KUKA KRL program: MyProgram_119().src

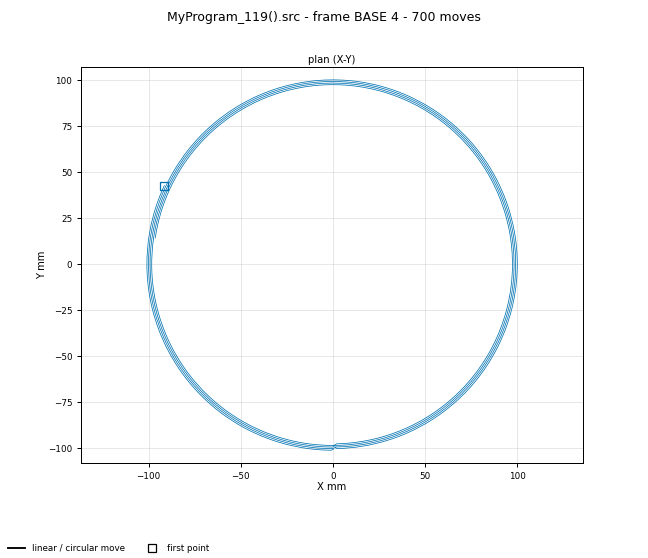
[picture p0: tool path of MyProgram_119().src in frame BASE 4, 700 of 700 moves have a stored position in this frame; points joined in program order, loops and branches not executed]
&ACCESS RVP
&REL 1
&PARAM TEMPLATE = C:\KRC\Roboter\Template\vorgabe
&PARAM EDITMASK = *
DEF MyProgram_119()
; ---- Setting reference (Base) ----
$BASE = BASE_DATA[4]

; --------------------------
; ---- Setting tool (TCP) ----
$TOOL = TOOL_DATA[3]
; --------------------------

$VEL.CP = VEL_APROX_PRINT
Startdeposition()
$VEL.CP = VEL_PRINT
LIN {X -91.493,Y 42.7067,Z 101,A 150.6977,B 24.9258,C -1.9891,E1 24.8544,E2 294.7155} C_DIS
LIN {X -92.8066,Y 39.7749,Z 101,A 152.6178,B 24.926,C -1.9868,E1 24.8522,E2 292.79} C_DIS
LIN {X -93.9596,Y 36.9649,Z 101,A 154.2845,B 24.9265,C -1.9796,E1 24.8505,E2 291.1312} C_DIS
LIN {X -95.1822,Y 33.6934,Z 101,A 156.3544,B 24.9268,C -1.9765,E1 24.8485,E2 289.0571} C_DIS
LIN {X -96.2277,Y 30.5829,Z 101,A 158.5957,B 24.9262,C -1.9837,E1 24.8466,E2 286.7858} C_DIS
LIN {X -97.2713,Y 27.0799,Z 101,A 160.5089,B 24.9271,C -1.9716,E1 24.8451,E2 284.8903} C_DIS
LIN {X -98.522,Y 22.1039,Z 101,A 163.2579,B 24.9282,C -1.9568,E1 24.8434,E2 282.1606} C_DIS
LIN {X -99.102,Y 19.3303,Z 101,A 165.2055,B 24.9277,C -1.9633,E1 24.8423,E2 280.1859} C_DIS
LIN {X -99.9373,Y 14.4011,Z 101,A 167.61,B 24.9295,C -1.9393,E1 24.8413,E2 277.8242} C_DIS
LIN {X -100.2963,Y 11.6391,Z 101,A 169.6473,B 24.9287,C -1.9499,E1 24.8406,E2 275.7496} C_DIS
LIN {X -100.8986,Y 3.8154,Z 101,A 173.661,B 24.9309,C -1.9204,E1 24.8399,E2 271.782} C_DIS
LIN {X -100.9502,Y -1.9696,Z 101,A 177.1716,B 24.9311,C -1.9176,E1 24.8399,E2 268.257} C_DIS
LIN {X -100.7114,Y -7.2249,Z 101,A 179.6583,B 24.933,C -1.891,E1 24.8402,E2 265.8188} C_DIS
LIN {X -100.1169,Y -13.0935,Z 101,A -176.3946,B 24.9323,C -1.9008,E1 24.8414,E2 261.8247} C_DIS
LIN {X -99.4794,Y -17.292,Z 101,A -174.1202,B 24.9331,C -1.8886,E1 24.8424,E2 259.566} C_DIS
LIN {X -98.8843,Y -20.4137,Z 101,A -172.2959,B 24.9335,C -1.8837,E1 24.8434,E2 257.7426} C_DIS
LIN {X -98.0917,Y -23.9337,Z 101,A -170.2804,B 24.934,C -1.8763,E1 24.8447,E2 255.733} C_DIS
LIN {X -97.2543,Y -27.1399,Z 101,A -168.3863,B 24.9344,C -1.871,E1 24.8461,E2 253.8404} C_DIS
LIN {X -95.3072,Y -33.3371,Z 101,A -164.6672,B 24.9351,C -1.8611,E1 24.8493,E2 250.1237} C_DIS
LIN {X -93.8132,Y -37.3364,Z 101,A -162.0084,B 24.935,C -1.8621,E1 24.852,E2 247.4474} C_DIS
LIN {X -91.5082,Y -42.6739,Z 101,A -158.9614,B 24.9363,C -1.844,E1 24.8554,E2 244.427} C_DIS
LIN {X -89.9932,Y -45.7829,Z 101,A -156.9304,B 24.9365,C -1.8409,E1 24.8579,E2 242.3925} C_DIS
LIN {X -88.288,Y -48.9909,Z 101,A -154.8266,B 24.9368,C -1.8367,E1 24.8607,E2 240.2874} C_DIS
LIN {X -85.444,Y -53.7984,Z 101,A -151.8215,B 24.9377,C -1.8226,E1 24.865,E2 237.3006} C_DIS
LIN {X -83.1904,Y -57.2225,Z 101,A -149.2876,B 24.9377,C -1.8239,E1 24.869,E2 234.751} C_DIS
LIN {X -81.3627,Y -59.7909,Z 101,A -147.5016,B 24.938,C -1.8194,E1 24.8719,E2 232.967} C_DIS
LIN {X -79.3097,Y -62.4885,Z 101,A -145.5763,B 24.9383,C -1.8148,E1 24.8752,E2 231.0434} C_DIS
LIN {X -77.0494,Y -65.2555,Z 101,A -143.6749,B 24.9389,C -1.8056,E1 24.8785,E2 229.1552} C_DIS
LIN {X -73.7308,Y -68.983,Z 101,A -140.7273,B 24.939,C -1.8033,E1 24.8841,E2 226.1999} C_DIS
LIN {X -71.3796,Y -71.4151,Z 101,A -138.9011,B 24.9396,C -1.7959,E1 24.8876,E2 224.3837} C_DIS
LIN {X -69.3421,Y -73.393,Z 101,A -137.1004,B 24.9393,C -1.7993,E1 24.8913,E2 222.5673} C_DIS
LIN {X -66.913,Y -75.6161,Z 101,A -134.6373,B 24.9381,C -1.817,E1 24.8966,E2 220.0524} C_DIS
LIN {X -63.8127,Y -78.2486,Z 101,A -132.5208,B 24.9389,C -1.8058,E1 24.9011,E2 217.9546} C_DIS
LIN {X -61.117,Y -80.3733,Z 101,A -131.0124,B 24.9402,C -1.7864,E1 24.9043,E2 216.4868} C_DIS
LIN {X -58.1677,Y -82.5329,Z 101,A -128.8413,B 24.9402,C -1.7864,E1 24.9093,E2 214.3081} C_DIS
LIN {X -54.8555,Y -84.7693,Z 101,A -126.6695,B 24.9407,C -1.7793,E1 24.9143,E2 212.146} C_DIS
LIN {X -50.7449,Y -87.292,Z 101,A -123.4729,B 24.9398,C -1.7921,E1 24.9221,E2 208.9093} C_DIS
LIN {X -47.8522,Y -88.9106,Z 101,A -121.9794,B 24.9409,C -1.7754,E1 24.9257,E2 207.4513} C_DIS
LIN {X -45.4378,Y -90.1696,Z 101,A -120.33,B 24.9409,C -1.7772,E1 24.9298,E2 205.7931} C_DIS
LIN {X -41.9811,Y -91.8297,Z 101,A -118.2406,B 24.9412,C -1.7715,E1 24.935,E2 203.712} C_DIS
LIN {X -38.9897,Y -93.1379,Z 101,A -116.4085,B 24.9414,C -1.7688,E1 24.9397,E2 201.882} C_DIS
LIN {X -34.2328,Y -94.9895,Z 101,A -113.3032,B 24.941,C -1.7739,E1 24.9479,E2 198.7582} C_DIS
LIN {X -30.1552,Y -96.3615,Z 101,A -111.3711,B 24.9424,C -1.7531,E1 24.9529,E2 196.872} C_DIS
LIN {X -26.5243,Y -97.4234,Z 101,A -108.3775,B 24.9404,C -1.7833,E1 24.9612,E2 193.8019} C_DIS
LIN {X -22.855,Y -98.3488,Z 101,A -106.897,B 24.9421,C -1.7571,E1 24.965,E2 192.3815} C_DIS
LIN {X -16.9752,Y -99.5327,Z 101,A -103.5642,B 24.9424,C -1.7531,E1 24.9742,E2 189.0547} C_DIS
LIN {X -13.0619,Y -100.121,Z 101,A -101.1076,B 24.9419,C -1.7605,E1 24.981,E2 186.5785} C_DIS
LIN {X -9.5303,Y -100.5189,Z 101,A -99.1069,B 24.9419,C -1.7597,E1 24.9865,E2 184.5785} C_DIS
LIN {X -5.5002,Y -100.8195,Z 101,A -96.5488,B 24.9413,C -1.7698,E1 24.9937,E2 181.9954} C_DIS
LIN {X -0.9129,Y -100.9657,Z 101,A -94.2262,B 24.942,C -1.7595,E1 25.0002,E2 179.6972} C_DIS
LIN {X -0.9129,Y -100.9657,Z 101,A -94.2262,B 24.942,C -1.7595,E1 25.0002,E2 179.6972} C_DIS
Enddeposition()
LIN {X 0.7006,Y -100.097,Z 101,A -94.1894,B 24.9431,C -1.7417,E1 25.0002,E2 179.7026} C_DIS
Startdeposition()
$VEL.CP = VEL_PRINT
LIN {X -2.9837,Y -100.0551,Z 101,A -96.3968,B 24.9434,C -1.7377,E1 24.9939,E2 181.9196} C_DIS
LIN {X -8.2546,Y -99.759,Z 101,A -99.1397,B 24.9427,C -1.748,E1 24.9864,E2 184.6391} C_DIS
LIN {X -10.6456,Y -99.5321,Z 101,A -100.6356,B 24.943,C -1.7436,E1 24.9822,E2 186.1463} C_DIS
LIN {X -16.0258,Y -98.8096,Z 101,A -104.2786,B 24.9443,C -1.7247,E1 24.972,E2 189.8371} C_DIS
LIN {X -19.3833,Y -98.2058,Z 101,A -105.6359,B 24.9428,C -1.7472,E1 24.9684,E2 191.1426} C_DIS
LIN {X -21.9592,Y -97.663,Z 101,A -107.9018,B 24.9445,C -1.7203,E1 24.9621,E2 193.4751} C_DIS
LIN {X -25.8197,Y -96.7127,Z 101,A -109.6986,B 24.9433,C -1.739,E1 24.9573,E2 195.2303} C_DIS
LIN {X -30.2063,Y -95.435,Z 101,A -112.2271,B 24.943,C -1.7439,E1 24.9506,E2 197.7513} C_DIS
LIN {X -35.0024,Y -93.7802,Z 101,A -115.2233,B 24.943,C -1.7432,E1 24.9427,E2 200.7553} C_DIS
LIN {X -39.1334,Y -92.1335,Z 101,A -117.5532,B 24.9424,C -1.7534,E1 24.9367,E2 203.066} C_DIS
LIN {X -42.6063,Y -90.5803,Z 101,A -119.8193,B 24.9424,C -1.7527,E1 24.9309,E2 205.3393} C_DIS
LIN {X -45.6761,Y -89.0709,Z 101,A -121.6953,B 24.9421,C -1.7581,E1 24.9263,E2 207.2076} C_DIS
LIN {X -48.5502,Y -87.5379,Z 101,A -124.3798,B 24.9438,C -1.7317,E1 24.9195,E2 209.9625} C_DIS
LIN {X -52.3977,Y -85.2915,Z 101,A -126.098,B 24.9416,C -1.7646,E1 24.9156,E2 211.6076} C_DIS
LIN {X -55.2394,Y -83.4779,Z 101,A -128.0767,B 24.9416,C -1.7659,E1 24.9109,E2 213.5897} C_DIS
LIN {X -57.5637,Y -81.8939,Z 101,A -129.9662,B 24.942,C -1.7588,E1 24.9066,E2 215.5026} C_DIS
LIN {X -60.5866,Y -79.6839,Z 101,A -132.7293,B 24.9432,C -1.741,E1 24.9003,E2 218.3179} C_DIS
LIN {X -64.2306,Y -76.7742,Z 101,A -134.8539,B 24.9416,C -1.7649,E1 24.8958,E2 220.3938} C_DIS
LIN {X -67.9037,Y -73.5466,Z 101,A -137.4269,B 24.9407,C -1.7782,E1 24.8905,E2 222.9453} C_DIS
LIN {X -70.1968,Y -71.3609,Z 101,A -139.231,B 24.9405,C -1.7823,E1 24.8869,E2 224.7471} C_DIS
LIN {X -72.61,Y -68.9051,Z 101,A -141.3632,B 24.9405,C -1.781,E1 24.8828,E2 226.8917} C_DIS
LIN {X -76.3774,Y -64.703,Z 101,A -144.5016,B 24.9398,C -1.7915,E1 24.877,E2 230.0192} C_DIS
LIN {X -78.6568,Y -61.9118,Z 101,A -146.6049,B 24.9396,C -1.795,E1 24.8733,E2 232.124} C_DIS
LIN {X -80.6494,Y -59.2928,Z 101,A -148.3867,B 24.9391,C -1.8031,E1 24.8703,E2 233.8951} C_DIS
LIN {X -82.5834,Y -56.5702,Z 101,A -150.8268,B 24.9399,C -1.79,E1 24.8664,E2 236.3785} C_DIS
LIN {X -84.496,Y -53.671,Z 101,A -152.1216,B 24.938,C -1.8186,E1 24.8645,E2 237.6116} C_DIS
LIN {X -86.627,Y -50.1577,Z 101,A -154.4412,B 24.9375,C -1.826,E1 24.8612,E2 239.9256} C_DIS
LIN {X -88.6618,Y -46.4655,Z 101,A -157.1228,B 24.9377,C -1.8234,E1 24.8576,E2 242.6275} C_DIS
LIN {X -90.0555,Y -43.7045,Z 101,A -159.0063,B 24.9377,C -1.8245,E1 24.8553,E2 244.5186} C_DIS
LIN {X -91.9197,Y -39.634,Z 101,A -162.5269,B 24.9393,C -1.7999,E1 24.8513,E2 248.1171} C_DIS
LIN {X -93.9682,Y -34.4956,Z 101,A -165.82,B 24.9389,C -1.8051,E1 24.8481,E2 251.4166} C_DIS
LIN {X -95.8576,Y -28.8337,Z 101,A -167.8821,B 24.9351,C -1.8603,E1 24.8465,E2 253.3587} C_DIS
LIN {X -96.5103,Y -26.569,Z 101,A -169.4978,B 24.9355,C -1.8555,E1 24.8452,E2 254.9954} C_DIS
LIN {X -97.3864,Y -23.155,Z 101,A -171.6399,B 24.9353,C -1.8575,E1 24.8438,E2 257.1453} C_DIS
LIN {X -98.2035,Y -19.3963,Z 101,A -173.8412,B 24.9348,C -1.8644,E1 24.8425,E2 259.3431} C_DIS
LIN {X -98.8363,Y -15.862,Z 101,A -176.063,B 24.9348,C -1.8653,E1 24.8415,E2 261.576} C_DIS
LIN {X -99.2655,Y -12.8949,Z 101,A -178.3144,B 24.9356,C -1.8531,E1 24.8407,E2 263.87} C_DIS
LIN {X -99.7582,Y -8.2647,Z 101,A -179.9211,B 24.9326,C -1.8966,E1 24.8403,E2 265.3825} C_DIS
LIN {X -100.0729,Y -2.3714,Z 101,A 175.9269,B 24.9336,C -1.8817,E1 24.8398,E2 269.595} C_DIS
LIN {X -100.0954,Y 0.9959,Z 101,A 174.3514,B 24.9324,C -1.8995,E1 24.8398,E2 271.1374} C_DIS
LIN {X -99.9873,Y 4.7622,Z 101,A 171.7367,B 24.9329,C -1.8914,E1 24.8401,E2 273.7873} C_DIS
LIN {X -99.7433,Y 8.4515,Z 101,A 169.9451,B 24.9317,C -1.9089,E1 24.8405,E2 275.548} C_DIS
LIN {X -99.2648,Y 12.9005,Z 101,A 167.5862,B 24.9306,C -1.9238,E1 24.8413,E2 277.8853} C_DIS
LIN {X -98.8225,Y 15.9485,Z 101,A 165.8016,B 24.9303,C -1.9287,E1 24.842,E2 279.6688} C_DIS
LIN {X -97.8958,Y 20.8933,Z 101,A 162.6806,B 24.9302,C -1.93,E1 24.8437,E2 282.8052} C_DIS
LIN {X -96.9348,Y 24.9712,Z 101,A 160.2729,B 24.9296,C -1.9373,E1 24.8454,E2 285.2096} C_DIS
LIN {X -95.5364,Y 29.8792,Z 101,A 157.2634,B 24.9292,C -1.9435,E1 24.8478,E2 288.2216} C_DIS
LIN {X -93.8825,Y 34.7305,Z 101,A 154.4878,B 24.9281,C -1.9579,E1 24.8503,E2 290.9787} C_DIS
LIN {X -92.1093,Y 39.1904,Z 101,A 151.9333,B 24.927,C -1.9727,E1 24.853,E2 293.5121} C_DIS
LIN {X -91.0749,Y 41.539,Z 101,A 150.4396,B 24.9268,C -1.9763,E1 24.8547,E2 295.0054} C_DIS
LIN {X -89.832,Y 44.1616,Z 101,A 148.0741,B 24.9281,C -1.9579,E1 24.8577,E2 297.4276} C_DIS
LIN {X -88.0636,Y 47.5894,Z 101,A 145.8824,B 24.9276,C -1.9649,E1 24.8606,E2 299.6142} C_DIS
LIN {X -86.2144,Y 50.8626,Z 101,A 144.331,B 24.9257,C -1.991,E1 24.8627,E2 301.1113} C_DIS
LIN {X -84.1782,Y 54.1661,Z 101,A 141.6968,B 24.9262,C -1.9835,E1 24.8666,E2 303.7768} C_DIS
LIN {X -80.2524,Y 59.8291,Z 101,A 137.9554,B 24.9249,C -2.0011,E1 24.8727,E2 307.4945} C_DIS
LIN {X -77.5079,Y 63.3449,Z 101,A 135.1326,B 24.9251,C -1.9988,E1 24.8776,E2 310.3361} C_DIS
LIN {X -73.9412,Y 67.4737,Z 101,A 132.0295,B 24.9244,C -2.0074,E1 24.8834,E2 313.4326} C_DIS
LIN {X -71.0995,Y 70.4614,Z 101,A 129.7788,B 24.9237,C -2.0168,E1 24.8877,E2 315.6704} C_DIS
LIN {X -67.7192,Y 73.7159,Z 101,A 127.0704,B 24.9233,C -2.0224,E1 24.8932,E2 318.3767} C_DIS
LIN {X -63.4929,Y 77.3882,Z 101,A 124.1903,B 24.9219,C -2.0406,E1 24.8993,E2 321.2246} C_DIS
LIN {X -61.4928,Y 78.9855,Z 101,A 122.181,B 24.9231,C -2.0252,E1 24.9038,E2 323.278} C_DIS
LIN {X -57.0068,Y 82.281,Z 101,A 119.1357,B 24.9222,C -2.0365,E1 24.9107,E2 326.307} C_DIS
LIN {X -53.02,Y 84.9047,Z 101,A 116.1874,B 24.9224,C -2.0342,E1 24.9177,E2 329.2701} C_DIS
LIN {X -50.0776,Y 86.673,Z 101,A 114.506,B 24.9214,C -2.0475,E1 24.9217,E2 330.925} C_DIS
LIN {X -46.541,Y 88.622,Z 101,A 112.3664,B 24.9206,C -2.0573,E1 24.9269,E2 333.0472} C_DIS
LIN {X -43.3756,Y 90.2135,Z 101,A 110.3409,B 24.9204,C -2.0607,E1 24.9319,E2 335.0701} C_DIS
LIN {X -39.8894,Y 91.8083,Z 101,A 107.6228,B 24.9215,C -2.0457,E1 24.939,E2 337.8301} C_DIS
LIN {X -36.6127,Y 93.1635,Z 101,A 106.2301,B 24.9196,C -2.0707,E1 24.9425,E2 339.1665} C_DIS
LIN {X -34.1586,Y 94.0911,Z 101,A 104.5603,B 24.9199,C -2.0668,E1 24.9469,E2 340.8491} C_DIS
LIN {X -31.2828,Y 95.0871,Z 101,A 103.0132,B 24.9192,C -2.0757,E1 24.9509,E2 342.3778} C_DIS
LIN {X -29.0314,Y 95.799,Z 101,A 101.4147,B 24.9198,C -2.0685,E1 24.9552,E2 343.9962} C_DIS
LIN {X -25.7437,Y 96.7332,Z 101,A 98.9755,B 24.9209,C -2.0536,E1 24.9619,E2 346.4746} C_DIS
LIN {X -22.1291,Y 97.6237,Z 101,A 97.5469,B 24.9188,C -2.0803,E1 24.9656,E2 347.8415} C_DIS
LIN {X -16.5738,Y 98.7179,Z 101,A 94.1038,B 24.9192,C -2.0757,E1 24.9751,E2 351.2994} C_DIS
LIN {X -10.1902,Y 99.5798,Z 101,A 90.7337,B 24.9181,C -2.0893,E1 24.9844,E2 354.6397} C_DIS
LIN {X -4.7667,Y 99.9871,Z 101,A 87.5182,B 24.9183,C -2.0868,E1 24.9934,E2 357.8622} C_DIS
LIN {X 0.5268,Y 100.0982,Z 101,A 84.3427,B 24.9187,C -2.0823,E1 25.0022,E2 361.0486} C_DIS
LIN {X 5.7674,Y 99.9336,Z 101,A 81.4712,B 24.9183,C -2.0873,E1 25.0102,E2 363.9076} C_DIS
LIN {X 8.3217,Y 99.7536,Z 101,A 79.1426,B 24.9207,C -2.0558,E1 25.0169,E2 366.3096} C_DIS
LIN {X 12.5536,Y 99.3097,Z 101,A 77.3041,B 24.9191,C -2.077,E1 25.0219,E2 368.0964} C_DIS
LIN {X 17.1869,Y 98.6145,Z 101,A 74.8657,B 24.9185,C -2.0851,E1 25.0285,E2 370.5131} C_DIS
LIN {X 22.4978,Y 97.5386,Z 101,A 71.4561,B 24.9195,C -2.0723,E1 25.0379,E2 373.9488} C_DIS
LIN {X 25.2776,Y 96.8561,Z 101,A 69.9253,B 24.9192,C -2.0753,E1 25.042,E2 375.4703} C_DIS
LIN {X 28.795,Y 95.8691,Z 101,A 67.4467,B 24.9205,C -2.0594,E1 25.0487,E2 377.9821} C_DIS
LIN {X 31.9491,Y 94.864,Z 101,A 65.7801,B 24.9199,C -2.0663,E1 25.0531,E2 379.6292} C_DIS
LIN {X 35.3881,Y 93.6355,Z 101,A 63.9232,B 24.9194,C -2.0731,E1 25.0579,E2 381.4662} C_DIS
LIN {X 38.949,Y 92.2112,Z 101,A 61.8875,B 24.9191,C -2.0768,E1 25.0632,E2 383.4884} C_DIS
LIN {X 41.1192,Y 91.2641,Z 101,A 60.5769,B 24.9191,C -2.077,E1 25.0665,E2 384.7954} C_DIS
LIN {X 43.6247,Y 90.0938,Z 101,A 58.7276,B 24.92,C -2.065,E1 25.0712,E2 386.6683} C_DIS
LIN {X 49.68,Y 86.9015,Z 101,A 54.9069,B 24.9202,C -2.0634,E1 25.0806,E2 390.4819} C_DIS
LIN {X 52.4585,Y 85.2543,Z 101,A 53.0967,B 24.9202,C -2.0621,E1 25.0849,E2 392.2895} C_DIS
LIN {X 54.5736,Y 83.9166,Z 101,A 51.4144,B 24.9212,C -2.0503,E1 25.0889,E2 393.9942} C_DIS
LIN {X 57.9099,Y 81.6483,Z 101,A 49.2842,B 24.9209,C -2.0533,E1 25.0938,E2 396.11} C_DIS
LIN {X 60.6655,Y 79.6236,Z 101,A 46.6029,B 24.9233,C -2.0222,E1 25.0999,E2 398.8552} C_DIS
LIN {X 64.1859,Y 76.8125,Z 101,A 44.8781,B 24.9212,C -2.05,E1 25.1034,E2 400.5077} C_DIS
LIN {X 66.6943,Y 74.6445,Z 101,A 42.9433,B 24.9216,C -2.0448,E1 25.1075,E2 402.4471} C_DIS
LIN {X 69.2792,Y 72.2522,Z 101,A 40.8642,B 24.9221,C -2.0382,E1 25.1118,E2 404.5332} C_DIS
LIN {X 71.9424,Y 69.6006,Z 101,A 38.7499,B 24.9223,C -2.035,E1 25.1159,E2 406.646} C_DIS
LIN {X 74.5803,Y 66.766,Z 101,A 36.5814,B 24.9226,C -2.0319,E1 25.12,E2 408.8123} C_DIS
LIN {X 76.207,Y 64.9031,Z 101,A 35.1815,B 24.9228,C -2.0293,E1 25.1225,E2 410.2122} C_DIS
LIN {X 78.6359,Y 61.9382,Z 101,A 33.0135,B 24.9231,C -2.0251,E1 25.1263,E2 412.38} C_DIS
LIN {X 80.7719,Y 59.1254,Z 101,A 30.763,B 24.9242,C -2.0111,E1 25.1301,E2 414.6527} C_DIS
LIN {X 83.494,Y 55.2149,Z 101,A 28.2001,B 24.9242,C -2.0106,E1 25.1341,E2 417.2041} C_DIS
LIN {X 85.5275,Y 52.0093,Z 101,A 26.0772,B 24.9245,C -2.0069,E1 25.1373,E2 419.3251} C_DIS
LIN {X 88.4343,Y 46.8975,Z 101,A 23.0136,B 24.9243,C -2.0097,E1 25.1414,E2 422.3661} C_DIS
LIN {X 90.4834,Y 42.8137,Z 101,A 19.9323,B 24.9262,C -1.9839,E1 25.1453,E2 425.4917} C_DIS
LIN {X 92.813,Y 37.4932,Z 101,A 17.0107,B 24.9257,C -1.9903,E1 25.1485,E2 428.3822} C_DIS
LIN {X 93.702,Y 35.2126,Z 101,A 15.3498,B 24.9268,C -1.9759,E1 25.1501,E2 430.068} C_DIS
LIN {X 94.8531,Y 31.9815,Z 101,A 13.5164,B 24.9268,C -1.9752,E1 25.1518,E2 431.8926} C_DIS
LIN {X 95.8353,Y 28.909,Z 101,A 11.2507,B 24.9285,C -1.9529,E1 25.1537,E2 434.198} C_DIS
LIN {X 97.7108,Y 21.7417,Z 101,A 7.6499,B 24.9276,C -1.9654,E1 25.1561,E2 437.7486} C_DIS
LIN {X 98.5163,Y 17.7329,Z 101,A 4.7673,B 24.9297,C -1.9364,E1 25.1577,E2 440.6826} C_DIS
LIN {X 99.0662,Y 14.3483,Z 101,A 2.5039,B 24.931,C -1.9183,E1 25.1586,E2 442.9755} C_DIS
LIN {X 99.5773,Y 10.2143,Z 101,A 1.336,B 24.928,C -1.9594,E1 25.1589,E2 444.0395} C_DIS
LIN {X 99.9111,Y 6.1631,Z 101,A -1.9506,B 24.9314,C -1.9133,E1 25.1596,E2 447.4153} C_DIS
LIN {X 100.0566,Y 2.9338,Z 101,A -3.848,B 24.9319,C -1.9055,E1 25.1598,E2 449.3198} C_DIS
LIN {X 100.0978,Y -0.6116,Z 101,A -5.3962,B 24.931,C -1.9182,E1 25.1598,E2 450.8289} C_DIS
LIN {X 100.0063,Y -4.3206,Z 101,A -7.9573,B 24.9328,C -1.8939,E1 25.1595,E2 453.4321} C_DIS
LIN {X 99.7945,Y -7.8104,Z 101,A -10.2974,B 24.9342,C -1.8739,E1 25.159,E2 455.8054} C_DIS
LIN {X 99.3001,Y -12.6283,Z 101,A -13.3909,B 24.9357,C -1.8523,E1 25.1578,E2 458.9317} C_DIS
LIN {X 98.3394,Y -18.6906,Z 101,A -15.4002,B 24.9323,C -1.901,E1 25.1569,E2 460.8144} C_DIS
LIN {X 97.2465,Y -23.7283,Z 101,A -18.6275,B 24.9337,C -1.8804,E1 25.155,E2 464.0716} C_DIS
LIN {X 96.3574,Y -27.1146,Z 101,A -21.8325,B 24.9375,C -1.8262,E1 25.1525,E2 467.3858} C_DIS
LIN {X 94.4759,Y -33.0791,Z 101,A -24.151,B 24.9348,C -1.8652,E1 25.1505,E2 469.5995} C_DIS
LIN {X 93.3391,Y -36.1656,Z 101,A -27.1789,B 24.9383,C -1.8138,E1 25.1473,E2 472.7318} C_DIS
LIN {X 91.0143,Y -41.6735,Z 101,A -29.3314,B 24.9356,C -1.8538,E1 25.145,E2 474.7781} C_DIS
LIN {X 89.3765,Y -45.0782,Z 101,A -32.0583,B 24.9376,C -1.8248,E1 25.1415,E2 477.5589} C_DIS
LIN {X 87.8167,Y -48.0446,Z 101,A -33.8804,B 24.9377,C -1.823,E1 25.1391,E2 479.3757} C_DIS
LIN {X 85.0848,Y -52.7316,Z 101,A -36.3481,B 24.9366,C -1.8395,E1 25.1357,E2 481.7918} C_DIS
LIN {X 82.1303,Y -57.2236,Z 101,A -39.399,B 24.9371,C -1.8319,E1 25.131,E2 484.8456} C_DIS
LIN {X 79.0604,Y -61.3964,Z 101,A -42.4573,B 24.9379,C -1.82,E1 25.1259,E2 487.9171} C_DIS
LIN {X 77.261,Y -63.6452,Z 101,A -44.5001,B 24.9393,C -1.8,E1 25.1222,E2 489.9977} C_DIS
LIN {X 74.6432,Y -66.6958,Z 101,A -46.5022,B 24.9389,C -1.8059,E1 25.1185,E2 491.9769} C_DIS
LIN {X 71.8665,Y -69.6793,Z 101,A -48.7723,B 24.9391,C -1.8026,E1 25.1142,E2 494.245} C_DIS
LIN {X 67.9034,Y -73.5469,Z 101,A -52.0245,B 24.9398,C -1.7917,E1 25.1076,E2 497.5094} C_DIS
LIN {X 65.5412,Y -75.6596,Z 101,A -54.039,B 24.9406,C -1.7796,E1 25.1033,E2 499.5444} C_DIS
LIN {X 61.9682,Y -78.6122,Z 101,A -57.3523,B 24.9427,C -1.7481,E1 25.096,E2 502.9197} C_DIS
LIN {X 57.8656,Y -81.6799,Z 101,A -58.7583,B 24.9392,C -1.8016,E1 25.0931,E2 504.1944} C_DIS
LIN {X 53.1117,Y -84.8474,Z 101,A -62.5262,B 24.9409,C -1.7755,E1 25.0842,E2 508.0115} C_DIS
LIN {X 50.3503,Y -86.5163,Z 101,A -64.7948,B 24.9422,C -1.7557,E1 25.0787,E2 510.3199} C_DIS
LIN {X 43.8916,Y -89.9656,Z 101,A -68.6624,B 24.9419,C -1.7611,E1 25.0691,E2 514.1639} C_DIS
LIN {X 38.9198,Y -92.2235,Z 101,A -72.2976,B 24.9435,C -1.7369,E1 25.0597,E2 517.8477} C_DIS
LIN {X 35.4642,Y -93.6067,Z 101,A -73.8684,B 24.9423,C -1.7553,E1 25.0557,E2 519.3713} C_DIS
LIN {X 32.0718,Y -94.8226,Z 101,A -77.1878,B 24.9455,C -1.7051,E1 25.0467,E2 522.803} C_DIS
LIN {X 25.9246,Y -96.6844,Z 101,A -79.6063,B 24.9427,C -1.7485,E1 25.0405,E2 525.1149} C_DIS
LIN {X 19.2144,Y -98.2386,Z 101,A -83.3099,B 24.9423,C -1.7539,E1 25.0304,E2 528.8007} C_DIS
LIN {X 12.1755,Y -99.3578,Z 101,A -87.46,B 24.9427,C -1.7482,E1 25.0189,E2 532.9603} C_DIS
LIN {X 5.8421,Y -99.9294,Z 101,A -91.7549,B 24.9444,C -1.722,E1 25.0068,E2 537.3153} C_DIS
LIN {X 2.2509,Y -100.0751,Z 101,A -93.3016,B 24.9432,C -1.7403,E1 25.0026,E2 538.8183} C_DIS
LIN {X 2.2509,Y -100.0751,Z 101,A -93.3016,B 24.9432,C -1.7403,E1 25.0026,E2 538.8183} C_DIS
Enddeposition()
LIN {X 0.6916,Y -99.2244,Z 101,A -93.6165,B 24.9408,C -1.7769,E1 25.002,E2 539.0464} C_DIS
Startdeposition()
$VEL.CP = VEL_PRINT
LIN {X 6.3538,Y -99.0267,Z 101,A -89.6742,B 24.9391,C -1.8033,E1 25.0131,E2 535.0428} C_DIS
LIN {X 12.1636,Y -98.4832,Z 101,A -86.8433,B 24.9403,C -1.7847,E1 25.0209,E2 532.2576} C_DIS
LIN {X 18.1451,Y -97.5584,Z 101,A -83.2608,B 24.9399,C -1.7906,E1 25.0308,E2 528.6648} C_DIS
LIN {X 23.6602,Y -96.3678,Z 101,A -80.0271,B 24.9398,C -1.7927,E1 25.0396,E2 525.4304} C_DIS
LIN {X 26.8003,Y -95.5424,Z 101,A -78.3328,B 24.9401,C -1.7878,E1 25.0441,E2 523.7505} C_DIS
LIN {X 31.9669,Y -93.9401,Z 101,A -74.9259,B 24.9391,C -1.8024,E1 25.0533,E2 520.3154} C_DIS
LIN {X 35.8208,Y -92.54,Z 101,A -71.783,B 24.9368,C -1.8358,E1 25.0617,E2 517.1001} C_DIS
LIN {X 40.3117,Y -90.6739,Z 101,A -69.7341,B 24.9386,C -1.8103,E1 25.0667,E2 515.1166} C_DIS
LIN {X 43.8065,Y -89.0372,Z 101,A -67.6711,B 24.9388,C -1.8074,E1 25.0719,E2 513.0657} C_DIS
LIN {X 45.9989,Y -87.9245,Z 101,A -66.2309,B 24.9385,C -1.8106,E1 25.0755,E2 511.6219} C_DIS
LIN {X 50.5879,Y -85.3664,Z 101,A -63.1025,B 24.9379,C -1.8198,E1 25.0831,E2 508.4812} C_DIS
LIN {X 55.554,Y -82.221,Z 101,A -59.8303,B 24.9379,C -1.8216,E1 25.0908,E2 505.2155} C_DIS
LIN {X 58.3914,Y -80.2313,Z 101,A -57.2713,B 24.936,C -1.8478,E1 25.0967,E2 502.6036} C_DIS
LIN {X 61.312,Y -78.0221,Z 101,A -55.6812,B 24.9371,C -1.8315,E1 25.1001,E2 501.0577} C_DIS
LIN {X 63.2853,Y -76.43,Z 101,A -53.8126,B 24.9358,C -1.8509,E1 25.1042,E2 499.1506} C_DIS
LIN {X 65.8199,Y -74.2598,Z 101,A -52.4995,B 24.9372,C -1.8309,E1 25.1068,E2 497.8899} C_DIS
LIN {X 69.8907,Y -70.4406,Z 101,A -49.0231,B 24.9359,C -1.8486,E1 25.1139,E2 494.3859} C_DIS
LIN {X 74.0098,Y -66.0992,Z 101,A -46.0025,B 24.9365,C -1.84,E1 25.1196,E2 491.399} C_DIS
LIN {X 77.5141,Y -61.9549,Z 101,A -42.4986,B 24.9349,C -1.8629,E1 25.1259,E2 487.8571} C_DIS
LIN {X 80.3128,Y -58.2802,Z 101,A -39.8563,B 24.9345,C -1.8691,E1 25.1303,E2 485.2127} C_DIS
LIN {X 82.4339,Y -55.2397,Z 101,A -37.3834,B 24.9331,C -1.8885,E1 25.1343,E2 482.7063} C_DIS
LIN {X 85.1675,Y -50.9244,Z 101,A -34.228,B 24.9319,C -1.9053,E1 25.1389,E2 479.5273} C_DIS
LIN {X 87.1332,Y -47.4804,Z 101,A -32.9116,B 24.9343,C -1.8727,E1 25.1406,E2 478.2946} C_DIS
LIN {X 88.6335,Y -44.6207,Z 101,A -30.6535,B 24.9328,C -1.894,E1 25.1435,E2 475.9982} C_DIS
LIN {X 90.1198,Y -41.5343,Z 101,A -28.7669,B 24.9326,C -1.8963,E1 25.1457,E2 474.1164} C_DIS
LIN {X 90.9993,Y -39.5686,Z 101,A -26.9002,B 24.9305,C -1.9254,E1 25.1479,E2 472.1913} C_DIS
LIN {X 92.5514,Y -35.7918,Z 101,A -25.096,B 24.9316,C -1.9101,E1 25.1497,E2 470.4331} C_DIS
LIN {X 93.7134,Y -32.6251,Z 101,A -22.5669,B 24.9294,C -1.9399,E1 25.152,E2 467.848} C_DIS
LIN {X 95.0254,Y -28.5807,Z 101,A -20.7534,B 24.9308,C -1.9215,E1 25.1535,E2 466.0883} C_DIS
LIN {X 96.026,Y -25.0129,Z 101,A -18.7831,B 24.9308,C -1.9215,E1 25.1549,E2 464.1295} C_DIS
LIN {X 96.6333,Y -22.5519,Z 101,A -16.8022,B 24.9289,C -1.9471,E1 25.1562,E2 462.0995} C_DIS
LIN {X 97.3395,Y -19.2831,Z 101,A -15.3945,B 24.93,C -1.932,E1 25.157,E2 460.7356} C_DIS
LIN {X 98.2316,Y -14.0393,Z 101,A -12.2896,B 24.9292,C -1.9432,E1 25.1584,E2 457.6224} C_DIS
LIN {X 98.6678,Y -10.5476,Z 101,A -10.5648,B 24.9296,C -1.9374,E1 25.1589,E2 455.9216} C_DIS
LIN {X 98.9435,Y -7.5412,Z 101,A -7.7728,B 24.9261,C -1.9856,E1 25.1596,E2 453.0325} C_DIS
LIN {X 99.1809,Y -3.1146,Z 101,A -6.001,B 24.9278,C -1.9618,E1 25.1598,E2 451.3274} C_DIS
LIN {X 99.1866,Y 2.929,Z 101,A -1.8322,B 24.925,C -2.0006,E1 25.1596,E2 447.0918} C_DIS
LIN {X 98.9706,Y 7.1841,Z 101,A 0.0102,B 24.9262,C -1.9834,E1 25.1592,E2 445.301} C_DIS
LIN {X 98.1834,Y 14.3784,Z 101,A 4.8169,B 24.9233,C -2.0221,E1 25.1575,E2 440.4314} C_DIS
LIN {X 97.4534,Y 18.6917,Z 101,A 6.5866,B 24.925,C -1.9993,E1 25.1567,E2 438.7256} C_DIS
LIN {X 96.75,Y 22.0468,Z 101,A 8.4021,B 24.925,C -1.9989,E1 25.1556,E2 436.9218} C_DIS
LIN {X 95.7769,Y 25.9485,Z 101,A 10.8729,B 24.9241,C -2.012,E1 25.1539,E2 434.4343} C_DIS
LIN {X 94.8252,Y 29.2361,Z 101,A 12.8188,B 24.9237,C -2.0168,E1 25.1523,E2 432.4882} C_DIS
LIN {X 93.8389,Y 32.2656,Z 101,A 14.7723,B 24.923,C -2.0268,E1 25.1506,E2 430.5221} C_DIS
LIN {X 92.5015,Y 35.9189,Z 101,A 16.6628,B 24.9236,C -2.0192,E1 25.1488,E2 428.6601} C_DIS
LIN {X 90.6665,Y 40.3278,Z 101,A 20.0236,B 24.9211,C -2.0512,E1 25.145,E2 425.242} C_DIS
LIN {X 88.5403,Y 44.8031,Z 101,A 22.5888,B 24.9214,C -2.0474,E1 25.1419,E2 422.6995} C_DIS
LIN {X 87.0559,Y 47.6229,Z 101,A 24.6266,B 24.9204,C -2.0603,E1 25.1391,E2 420.642} C_DIS
LIN {X 84.739,Y 51.632,Z 101,A 26.9269,B 24.921,C -2.0526,E1 25.1359,E2 418.3717} C_DIS
LIN {X 82.719,Y 54.8101,Z 101,A 29.0185,B 24.9208,C -2.055,E1 25.1327,E2 416.285} C_DIS
LIN {X 80.146,Y 58.5079,Z 101,A 31.7329,B 24.92,C -2.066,E1 25.1283,E2 413.5579} C_DIS
LIN {X 77.8797,Y 61.4922,Z 101,A 33.7179,B 24.92,C -2.0642,E1 25.125,E2 411.5865} C_DIS
LIN {X 75.911,Y 63.9093,Z 101,A 35.5946,B 24.9195,C -2.0714,E1 25.1216,E2 409.7013} C_DIS
LIN {X 74.3224,Y 65.75,Z 101,A 37.1035,B 24.919,C -2.0787,E1 25.1188,E2 408.182} C_DIS
LIN {X 72.0836,Y 68.1952,Z 101,A 39.0416,B 24.9186,C -2.0839,E1 25.1151,E2 406.24} C_DIS
LIN {X 69.5519,Y 70.7753,Z 101,A 41.1003,B 24.9183,C -2.0873,E1 25.111,E2 404.1822} C_DIS
LIN {X 66.9465,Y 73.2444,Z 101,A 43.1126,B 24.9181,C -2.0892,E1 25.1069,E2 402.1736} C_DIS
LIN {X 64.2983,Y 75.5796,Z 101,A 44.9423,B 24.9185,C -2.0851,E1 25.1031,E2 400.3607} C_DIS
LIN {X 61.0442,Y 78.2337,Z 101,A 47.66,B 24.9172,C -2.1009,E1 25.0971,E2 397.6159} C_DIS
LIN {X 57.9902,Y 80.5225,Z 101,A 49.7483,B 24.9172,C -2.1003,E1 25.0925,E2 395.5365} C_DIS
LIN {X 55.4221,Y 82.3104,Z 101,A 51.6178,B 24.9168,C -2.1057,E1 25.0881,E2 393.6605} C_DIS
LIN {X 52.9337,Y 83.933,Z 101,A 53.3745,B 24.9165,C -2.1099,E1 25.084,E2 391.8994} C_DIS
LIN {X 49.5448,Y 85.976,Z 101,A 55.2659,B 24.9174,C -2.0983,E1 25.0795,E2 390.0414} C_DIS
LIN {X 45.8575,Y 87.9989,Z 101,A 58.0416,B 24.9161,C -2.1148,E1 25.0726,E2 387.2347} C_DIS
LIN {X 42.9669,Y 89.4449,Z 101,A 59.7167,B 24.9165,C -2.1098,E1 25.0685,E2 385.5757} C_DIS
LIN {X 40.1177,Y 90.76,Z 101,A 61.6838,B 24.9159,C -2.1177,E1 25.0634,E2 383.5948} C_DIS
LIN {X 35.9128,Y 92.5039,Z 101,A 64.3228,B 24.9156,C -2.1208,E1 25.0566,E2 380.9544} C_DIS
LIN {X 32.6977,Y 93.688,Z 101,A 66.9189,B 24.9136,C -2.146,E1 25.0496,E2 378.304} C_DIS
LIN {X 28.5833,Y 95.0246,Z 101,A 68.7127,B 24.9156,C -2.1213,E1 25.045,E2 376.5719} C_DIS
LIN {X 25.5467,Y 95.8855,Z 101,A 70.5042,B 24.9156,C -2.1213,E1 25.0402,E2 374.7831} C_DIS
LIN {X 23.2273,Y 96.4734,Z 101,A 71.8399,B 24.9156,C -2.1204,E1 25.0365,E2 373.4516} C_DIS
LIN {X 19.4176,Y 97.3129,Z 101,A 74.2357,B 24.9152,C -2.1268,E1 25.03,E2 371.0438} C_DIS
LIN {X 15.8591,Y 97.9556,Z 101,A 76.7431,B 24.9139,C -2.1431,E1 25.023,E2 368.5002} C_DIS
LIN {X 12.4184,Y 98.4502,Z 101,A 78.364,B 24.915,C -2.1292,E1 25.0186,E2 366.9135} C_DIS
LIN {X 7.0075,Y 98.9825,Z 101,A 81.1509,B 24.916,C -2.1166,E1 25.0109,E2 364.1583} C_DIS
LIN {X 1.3541,Y 99.2216,Z 101,A 84.4602,B 24.9159,C -2.1178,E1 25.0017,E2 360.847} C_DIS
LIN {X -4.3687,Y 99.1336,Z 101,A 87.472,B 24.9168,C -2.1063,E1 24.9934,E2 357.8622} C_DIS
LIN {X -9.2517,Y 98.7976,Z 101,A 90.7224,B 24.9157,C -2.1203,E1 24.9842,E2 354.5773} C_DIS
LIN {X -14.0161,Y 98.2349,Z 101,A 93.5781,B 24.9156,C -2.1217,E1 24.9763,E2 351.7162} C_DIS
LIN {X -18.1165,Y 97.5636,Z 101,A 96.4336,B 24.9144,C -2.1363,E1 24.9683,E2 348.8232} C_DIS
LIN {X -21.3424,Y 96.9076,Z 101,A 97.7828,B 24.9161,C -2.1149,E1 24.9648,E2 347.5232} C_DIS
LIN {X -25.0619,Y 96.0134,Z 101,A 100.0596,B 24.9161,C -2.1152,E1 24.9586,E2 345.2425} C_DIS
LIN {X -28.7965,Y 94.9614,Z 101,A 102.5226,B 24.9157,C -2.1206,E1 24.9519,E2 342.7625} C_DIS
LIN {X -32.7072,Y 93.6846,Z 101,A 104.8611,B 24.916,C -2.1164,E1 24.9458,E2 340.4296} C_DIS
LIN {X -36.3507,Y 92.3319,Z 101,A 107.4865,B 24.9152,C -2.1269,E1 24.9389,E2 337.7736} C_DIS
LIN {X -39.6612,Y 90.9589,Z 101,A 108.9927,B 24.917,C -2.1041,E1 24.9351,E2 336.3183} C_DIS
LIN {X -42.4708,Y 89.6833,Z 101,A 111.0187,B 24.9165,C -2.1099,E1 24.9299,E2 334.2734} C_DIS
LIN {X -45.9858,Y 87.9314,Z 101,A 113.1082,B 24.9173,C -2.0999,E1 24.9248,E2 332.2019} C_DIS
LIN {X -48.7251,Y 86.444,Z 101,A 114.8934,B 24.9176,C -2.0963,E1 24.9204,E2 330.4202} C_DIS
LIN {X -53.1742,Y 83.7813,Z 101,A 117.9615,B 24.9178,C -2.0933,E1 24.9131,E2 327.3496} C_DIS
LIN {X -56.1482,Y 81.8185,Z 101,A 120.2897,B 24.9174,C -2.0987,E1 24.9077,E2 325.0009} C_DIS
LIN {X -61.7314,Y 77.6907,Z 101,A 123.9325,B 24.9191,C -2.0776,E1 24.8997,E2 321.3952} C_DIS
LIN {X -64.2208,Y 75.6457,Z 101,A 126.0114,B 24.9188,C -2.081,E1 24.8952,E2 319.3003} C_DIS
LIN {X -67.0993,Y 73.1042,Z 101,A 128.0301,B 24.9197,C -2.0691,E1 24.891,E2 317.3018} C_DIS
LIN {X -69.5965,Y 70.7312,Z 101,A 130.2343,B 24.9195,C -2.0717,E1 24.8866,E2 315.0822} C_DIS
LIN {X -72.5465,Y 67.703,Z 101,A 133.0859,B 24.9189,C -2.0797,E1 24.881,E2 312.1992} C_DIS
LIN {X -74.931,Y 65.0536,Z 101,A 135.4065,B 24.9186,C -2.0835,E1 24.8768,E2 309.8591} C_DIS
LIN {X -77.8049,Y 61.5869,Z 101,A 137.1334,B 24.9214,C -2.0468,E1 24.8739,E2 308.2114} C_DIS
LIN {X -81.0438,Y 57.2582,Z 101,A 140.4455,B 24.9216,C -2.0448,E1 24.8684,E2 304.8883} C_DIS
LIN {X -84.4996,Y 52.0259,Z 101,A 144.1518,B 24.9222,C -2.0374,E1 24.8628,E2 301.1807} C_DIS
LIN {X -86.4907,Y 48.6414,Z 101,A 147.2761,B 24.9204,C -2.06,E1 24.8584,E2 297.9862} C_DIS
LIN {X -88.9227,Y 44.0374,Z 101,A 149.3298,B 24.9236,C -2.0188,E1 24.8559,E2 296.0199} C_DIS
LIN {X -90.4317,Y 40.8491,Z 101,A 151.3862,B 24.924,C -2.0133,E1 24.8535,E2 293.9653} C_DIS
LIN {X -92.7186,Y 35.3533,Z 101,A 154.8262,B 24.9248,C -2.0029,E1 24.8499,E2 290.531} C_DIS
LIN {X -94.8443,Y 29.1746,Z 101,A 158.642,B 24.9256,C -1.9925,E1 24.8465,E2 286.7182} C_DIS
LIN {X -95.7548,Y 26.0305,Z 101,A 160.8806,B 24.9251,C -1.9982,E1 24.8448,E2 284.4529} C_DIS
LIN {X -96.9395,Y 21.196,Z 101,A 163.7449,B 24.9258,C -1.9887,E1 24.843,E2 281.5944} C_DIS
LIN {X -97.836,Y 16.5744,Z 101,A 166.1852,B 24.9272,C -1.9707,E1 24.8418,E2 279.1827} C_DIS
LIN {X -98.3354,Y 13.3046,Z 101,A 168.1772,B 24.9274,C -1.9673,E1 24.841,E2 277.187} C_DIS
LIN {X -98.7235,Y 10.0156,Z 101,A 170.0014,B 24.9281,C -1.9582,E1 24.8405,E2 275.3735} C_DIS
LIN {X -99.042,Y 6.1268,Z 101,A 172.2309,B 24.9287,C -1.9501,E1 24.84,E2 273.1499} C_DIS
LIN {X -99.1915,Y 2.768,Z 101,A 174.358,B 24.9287,C -1.9501,E1 24.8398,E2 271.01} C_DIS
LIN {X -99.2287,Y -0.4872,Z 101,A 176.3263,B 24.9289,C -1.947,E1 24.8398,E2 269.0372} C_DIS
LIN {X -99.0715,Y -5.6035,Z 101,A 179.0811,B 24.9301,C -1.9308,E1 24.8401,E2 266.3045} C_DIS
LIN {X -98.7771,Y -9.4735,Z 101,A -178.1706,B 24.9294,C -1.9407,E1 24.8408,E2 263.516} C_DIS
LIN {X -98.4142,Y -12.6963,Z 101,A -177.1328,B 24.9318,C -1.9068,E1 24.8411,E2 262.5531} C_DIS
LIN {X -98.0471,Y -15.2749,Z 101,A -175.2845,B 24.9314,C -1.9135,E1 24.8419,E2 260.6776} C_DIS
LIN {X -97.5178,Y -18.357,Z 101,A -173.3544,B 24.9314,C -1.9121,E1 24.8428,E2 258.7396} C_DIS
LIN {X -96.7804,Y -21.9152,Z 101,A -171.2355,B 24.9319,C -1.9063,E1 24.8441,E2 256.6221} C_DIS
LIN {X -95.9715,Y -25.2251,Z 101,A -169.2467,B 24.9323,C -1.9009,E1 24.8455,E2 254.6344} C_DIS
LIN {X -95.0127,Y -28.6236,Z 101,A -166.6437,B 24.9313,C -1.9139,E1 24.8476,E2 251.9853} C_DIS
LIN {X -93.8293,Y -32.2898,Z 101,A -164.9883,B 24.9332,C -1.888,E1 24.849,E2 250.3825} C_DIS
LIN {X -92.6985,Y -35.4063,Z 101,A -163.3101,B 24.9341,C -1.8743,E1 24.8506,E2 248.7273} C_DIS
LIN {X -90.9835,Y -39.6049,Z 101,A -160.4627,B 24.9341,C -1.8745,E1 24.8537,E2 245.8637} C_DIS
LIN {X -89.5953,Y -42.6539,Z 101,A -158.4712,B 24.9344,C -1.871,E1 24.856,E2 243.8698} C_DIS
LIN {X -88.1041,Y -45.6565,Z 101,A -156.4916,B 24.9347,C -1.8671,E1 24.8586,E2 241.8888} C_DIS
LIN {X -86.5603,Y -48.5169,Z 101,A -154.801,B 24.9355,C -1.8557,E1 24.8608,E2 240.2166} C_DIS
LIN {X -84.6236,Y -51.8218,Z 101,A -152.3532,B 24.9353,C -1.8579,E1 24.8643,E2 237.7508} C_DIS
LIN {X -81.9341,Y -55.9778,Z 101,A -149.5094,B 24.9358,C -1.85,E1 24.8687,E2 234.9115} C_DIS
LIN {X -80.1354,Y -58.5225,Z 101,A -147.7543,B 24.9363,C -1.844,E1 24.8716,E2 233.1621} C_DIS
LIN {X -77.4904,Y -61.9848,Z 101,A -145.1959,B 24.9366,C -1.8394,E1 24.876,E2 230.6025} C_DIS
LIN {X -75.579,Y -64.299,Z 101,A -142.6043,B 24.9348,C -1.8654,E1 24.8808,E2 227.9372} C_DIS
LIN {X -72.2921,Y -67.9735,Z 101,A -140.6224,B 24.9373,C -1.8288,E1 24.8844,E2 226.0338} C_DIS
LIN {X -69.7037,Y -70.6253,Z 101,A -138.4997,B 24.9377,C -1.8237,E1 24.8886,E2 223.9143} C_DIS
LIN {X -66.8615,Y -73.3224,Z 101,A -136.285,B 24.9381,C -1.8174,E1 24.8931,E2 221.7055} C_DIS
LIN {X -64.6554,Y -75.2749,Z 101,A -134.1342,B 24.9372,C -1.8299,E1 24.8977,E2 219.5165} C_DIS
LIN {X -60.0562,Y -78.9944,Z 101,A -131.0058,B 24.9384,C -1.8135,E1 24.9045,E2 216.4156} C_DIS
LIN {X -58.0196,Y -80.5015,Z 101,A -129.4374,B 24.9383,C -1.8148,E1 24.9081,E2 214.8387} C_DIS
LIN {X -53.2839,Y -83.7109,Z 101,A -126.1864,B 24.9388,C -1.8077,E1 24.9156,E2 211.594} C_DIS
LIN {X -49.0631,Y -86.2527,Z 101,A -123.527,B 24.9395,C -1.7969,E1 24.922,E2 208.952} C_DIS
LIN {X -46.5781,Y -87.6194,Z 101,A -121.8164,B 24.9395,C -1.7974,E1 24.9262,E2 207.2355} C_DIS
LIN {X -44.0863,Y -88.8985,Z 101,A -120.2311,B 24.9397,C -1.7942,E1 24.9301,E2 205.6535} C_DIS
LIN {X -41.0855,Y -90.3252,Z 101,A -118.0237,B 24.9391,C -1.8024,E1 24.9358,E2 203.4211} C_DIS
LIN {X -37.4294,Y -91.8998,Z 101,A -115.8956,B 24.9397,C -1.7939,E1 24.9412,E2 201.3084} C_DIS
LIN {X -31.965,Y -93.9407,Z 101,A -112.5499,B 24.9399,C -1.7901,E1 24.95,E2 197.9651} C_DIS
LIN {X -28.8738,Y -94.9375,Z 101,A -110.6482,B 24.9399,C -1.7896,E1 24.9551,E2 196.0612} C_DIS
LIN {X -26.599,Y -95.599,Z 101,A -109.342,B 24.9402,C -1.7865,E1 24.9586,E2 194.7602} C_DIS
LIN {X -22.6931,Y -96.6007,Z 101,A -106.9386,B 24.9401,C -1.7879,E1 24.9651,E2 192.35} C_DIS
LIN {X -19.4121,Y -97.314,Z 101,A -105.1829,B 24.9406,C -1.7804,E1 24.9699,E2 190.6102} C_DIS
LIN {X -16.0922,Y -97.9166,Z 101,A -103.4257,B 24.9411,C -1.7727,E1 24.9747,E2 188.8695} C_DIS
LIN {X -11.0263,Y -98.6166,Z 101,A -100.0346,B 24.9401,C -1.7883,E1 24.9842,E2 185.4389} C_DIS
LIN {X -4.6565,Y -99.1212,Z 101,A -96.5174,B 24.9405,C -1.7818,E1 24.9939,E2 181.9356} C_DIS
LIN {X 0.0011,Y -99.2315,Z 101,A -93.6455,B 24.94,C -1.7891,E1 25.002,E2 179.0464} C_DIS
LIN {X 0.0011,Y -99.2315,Z 101,A -93.6455,B 24.94,C -1.7891,E1 25.002,E2 179.0464} C_DIS
Enddeposition()
LIN {X 0.7034,Y -98.3509,Z 101,A -94.9046,B 24.943,C -1.7434,E1 24.9982,E2 180.4139} C_DIS
Startdeposition()
$VEL.CP = VEL_PRINT
LIN {X -3.7155,Y -98.291,Z 101,A -96.6585,B 24.9411,C -1.7726,E1 24.9935,E2 182.0988} C_DIS
LIN {X -9.1858,Y -97.9302,Z 101,A -99.8022,B 24.941,C -1.7743,E1 24.9847,E2 185.2394} C_DIS
LIN {X -12.3233,Y -97.5854,Z 101,A -101.8729,B 24.9415,C -1.7662,E1 24.9789,E2 187.3308} C_DIS
LIN {X -15.4933,Y -97.1332,Z 101,A -103.7927,B 24.9416,C -1.7647,E1 24.9736,E2 189.2559} C_DIS
LIN {X -18.9372,Y -96.5204,Z 101,A -105.7837,B 24.9415,C -1.7671,E1 24.9681,E2 191.2432} C_DIS
LIN {X -21.5107,Y -95.9806,Z 101,A -107.3656,B 24.9415,C -1.766,E1 24.9638,E2 192.8297} C_DIS
LIN {X -25.1637,Y -95.0876,Z 101,A -109.3058,B 24.9409,C -1.7762,E1 24.9586,E2 194.7485} C_DIS
LIN {X -28.0173,Y -94.2853,Z 101,A -111.0552,B 24.9409,C -1.7765,E1 24.9539,E2 196.4998} C_DIS
LIN {X -30.8873,Y -93.3862,Z 101,A -112.8397,B 24.9409,C -1.7767,E1 24.9491,E2 198.2873} C_DIS
LIN {X -36.5759,Y -91.3082,Z 101,A -116.5468,B 24.941,C -1.7735,E1 24.9394,E2 202.0094} C_DIS
LIN {X -39.5964,Y -90.0383,Z 101,A -118.4712,B 24.941,C -1.775,E1 24.9345,E2 203.9347} C_DIS
LIN {X -42.0856,Y -88.9034,Z 101,A -120.1217,B 24.941,C -1.7749,E1 24.9303,E2 205.5898} C_DIS
LIN {X -45.436,Y -87.2379,Z 101,A -122.007,B 24.9401,C -1.7879,E1 24.9257,E2 207.4493} C_DIS
LIN {X -47.9813,Y -85.8631,Z 101,A -123.919,B 24.9405,C -1.7823,E1 24.9209,E2 209.38} C_DIS
LIN {X -50.916,Y -84.1563,Z 101,A -125.881,B 24.9402,C -1.7857,E1 24.9162,E2 211.3399} C_DIS
LIN {X -52.849,Y -82.9564,Z 101,A -127.3538,B 24.9404,C -1.7826,E1 24.9127,E2 212.8247} C_DIS
LIN {X -56.2152,Y -80.7127,Z 101,A -129.4359,B 24.9396,C -1.7959,E1 24.908,E2 214.8822} C_DIS
LIN {X -58.7412,Y -78.8944,Z 101,A -131.18,B 24.9392,C -1.8013,E1 24.904,E2 216.6195} C_DIS
LIN {X -62.2617,Y -76.1468,Z 101,A -134.629,B 24.9408,C -1.7772,E1 24.8964,E2 220.1386} C_DIS
LIN {X -65.2701,Y -73.5846,Z 101,A -136.565,B 24.9397,C -1.7941,E1 24.8924,E2 222.0422} C_DIS
LIN {X -68.2375,Y -70.8401,Z 101,A -138.7304,B 24.9389,C -1.8053,E1 24.888,E2 224.1898} C_DIS
LIN {X -70.8399,Y -68.2377,Z 101,A -140.7367,B 24.9383,C -1.8146,E1 24.8841,E2 226.1826} C_DIS
LIN {X -75.2979,Y -63.2866,Z 101,A -144.5929,B 24.9376,C -1.8241,E1 24.877,E2 230.0333} C_DIS
LIN {X -76.6405,Y -61.6526,Z 101,A -146.2541,B 24.9384,C -1.8126,E1 24.874,E2 231.7296} C_DIS
LIN {X -79.222,Y -58.2976,Z 101,A -148.2581,B 24.9369,C -1.8341,E1 24.8707,E2 233.6921} C_DIS
LIN {X -80.4418,Y -56.6049,Z 101,A -149.6789,B 24.9372,C -1.8302,E1 24.8684,E2 235.129} C_DIS
LIN {X -82.2162,Y -53.9926,Z 101,A -151.5058,B 24.9369,C -1.8353,E1 24.8655,E2 236.9529} C_DIS
LIN {X -84.0028,Y -51.1684,Z 101,A -153.4645,B 24.9365,C -1.84,E1 24.8626,E2 238.9103} C_DIS
LIN {X -85.7702,Y -48.1476,Z 101,A -155.5408,B 24.9362,C -1.8443,E1 24.8597,E2 240.9873} C_DIS
LIN {X -87.0626,Y -45.7689,Z 101,A -157.2053,B 24.9362,C -1.8457,E1 24.8576,E2 242.6574} C_DIS
LIN {X -88.4277,Y -43.0754,Z 101,A -158.7362,B 24.9353,C -1.8581,E1 24.8557,E2 244.1668} C_DIS
LIN {X -89.3618,Y -41.1016,Z 101,A -160.2009,B 24.9355,C -1.8553,E1 24.8539,E2 245.6461} C_DIS
LIN {X -90.8486,Y -37.7028,Z 101,A -162.3396,B 24.935,C -1.8623,E1 24.8516,E2 247.7802} C_DIS
LIN {X -91.9833,Y -34.839,Z 101,A -164.1827,B 24.9347,C -1.8659,E1 24.8497,E2 249.6249} C_DIS
LIN {X -93.6306,Y -30.1333,Z 101,A -167.1855,B 24.9344,C -1.8713,E1 24.847,E2 252.6318} C_DIS
LIN {X -94.4697,Y -27.3957,Z 101,A -168.8734,B 24.934,C -1.8757,E1 24.8457,E2 254.3191} C_DIS
LIN {X -95.451,Y -23.7481,Z 101,A -171.011,B 24.9334,C -1.8845,E1 24.8442,E2 256.4483} C_DIS
LIN {X -96.1153,Y -20.8933,Z 101,A -172.7092,B 24.933,C -1.8901,E1 24.8432,E2 258.143} C_DIS
LIN {X -96.715,Y -17.9208,Z 101,A -174.5631,B 24.9328,C -1.8927,E1 24.8422,E2 260.0016} C_DIS
LIN {X -97.3258,Y -14.2311,Z 101,A -176.7146,B 24.9323,C -1.9005,E1 24.8413,E2 262.1475} C_DIS
LIN {X -97.7801,Y -10.6735,Z 101,A -178.833,B 24.9319,C -1.9061,E1 24.8406,E2 264.265} C_DIS
LIN {X -98.1021,Y -7.1347,Z 101,A 179.0737,B 24.9315,C -1.912,E1 24.8401,E2 266.357} C_DIS
LIN {X -98.2566,Y -4.5161,Z 101,A 177.6793,B 24.9308,C -1.9212,E1 24.8399,E2 267.7377} C_DIS
LIN {X -98.355,Y -1.1049,Z 101,A 175.5213,B 24.9308,C -1.922,E1 24.8398,E2 269.9067} C_DIS
LIN {X -98.3255,Y 2.6307,Z 101,A 173.3572,B 24.9302,C -1.9295,E1 24.8398,E2 272.0662} C_DIS
LIN {X -98.155,Y 6.3522,Z 101,A 171.5211,B 24.9289,C -1.9473,E1 24.8401,E2 273.8707} C_DIS
LIN {X -98.0028,Y 8.3932,Z 101,A 169.9369,B 24.9296,C -1.9384,E1 24.8405,E2 275.4858} C_DIS
LIN {X -97.7157,Y 11.2407,Z 101,A 168.4669,B 24.9287,C -1.9502,E1 24.8409,E2 276.9364} C_DIS
LIN {X -97.17,Y 15.2554,Z 101,A 165.8692,B 24.9287,C -1.9501,E1 24.842,E2 279.5499} C_DIS
LIN {X -96.4775,Y 19.1597,Z 101,A 163.4905,B 24.9283,C -1.9552,E1 24.8432,E2 281.9304} C_DIS
LIN {X -95.613,Y 23.0842,Z 101,A 160.6091,B 24.9291,C -1.9452,E1 24.8451,E2 284.8524} C_DIS
LIN {X -94.5501,Y 27.1119,Z 101,A 158.9401,B 24.9267,C -1.9773,E1 24.8463,E2 286.4545} C_DIS
LIN {X -93.2308,Y 31.3482,Z 101,A 156.2894,B 24.9263,C -1.9833,E1 24.8486,E2 289.1064} C_DIS
LIN {X -92.059,Y 34.6389,Z 101,A 154.4241,B 24.9254,C -1.9951,E1 24.8503,E2 290.9539} C_DIS
LIN {X -90.5701,Y 38.3637,Z 101,A 151.7491,B 24.9257,C -1.9912,E1 24.8532,E2 293.6532} C_DIS
LIN {X -89.3333,Y 41.1629,Z 101,A 150.2603,B 24.9245,C -2.0061,E1 24.8548,E2 295.1145} C_DIS
LIN {X -88.0135,Y 43.9132,Z 101,A 147.9926,B 24.9253,C -1.9954,E1 24.8577,E2 297.42} C_DIS
LIN {X -85.9887,Y 47.7564,Z 101,A 145.9669,B 24.9235,C -2.0193,E1 24.8603,E2 299.3995} C_DIS
LIN {X -84.7002,Y 50.0055,Z 101,A 144.207,B 24.9238,C -2.0155,E1 24.8628,E2 301.1776} C_DIS
LIN {X -83.3813,Y 52.1751,Z 101,A 142.5739,B 24.9238,C -2.0146,E1 24.8652,E2 302.8211} C_DIS
LIN {X -80.7219,Y 56.2019,Z 101,A 139.3136,B 24.9244,C -2.0078,E1 24.8704,E2 306.1139} C_DIS
LIN {X -78.534,Y 59.221,Z 101,A 137.6147,B 24.9228,C -2.0291,E1 24.8731,E2 307.7702} C_DIS
LIN {X -76.8383,Y 61.4071,Z 101,A 135.4349,B 24.9239,C -2.0147,E1 24.877,E2 309.9945} C_DIS
LIN {X -74.3107,Y 64.4416,Z 101,A 133.6039,B 24.9223,C -2.036,E1 24.8803,E2 311.783} C_DIS
LIN {X -71.1302,Y 67.9359,Z 101,A 131.1297,B 24.921,C -2.0521,E1 24.8849,E2 314.2298} C_DIS
LIN {X -69.1647,Y 69.9351,Z 101,A 129.3243,B 24.9212,C -2.0503,E1 24.8885,E2 316.047} C_DIS
LIN {X -66.4793,Y 72.4926,Z 101,A 126.8186,B 24.9217,C -2.0439,E1 24.8937,E2 318.5782} C_DIS
LIN {X -62.5346,Y 75.9229,Z 101,A 124.2948,B 24.9198,C -2.0681,E1 24.8989,E2 321.0543} C_DIS
LIN {X -60.3632,Y 77.6604,Z 101,A 122.4278,B 24.9202,C -2.0633,E1 24.9031,E2 322.9395} C_DIS
LIN {X -57.4701,Y 79.825,Z 101,A 120.2846,B 24.9199,C -2.0663,E1 24.9079,E2 325.0831} C_DIS
LIN {X -54.7252,Y 81.7318,Z 101,A 118.4386,B 24.9194,C -2.0735,E1 24.9121,E2 326.9181} C_DIS
LIN {X -51.6549,Y 83.7062,Z 101,A 116.2018,B 24.9194,C -2.0738,E1 24.9174,E2 329.1614} C_DIS
LIN {X -48.5568,Y 85.5405,Z 101,A 114.0455,B 24.9192,C -2.0756,E1 24.9226,E2 331.3199} C_DIS
LIN {X -45.0463,Y 87.4392,Z 101,A 112.0727,B 24.918,C -2.0914,E1 24.9274,E2 333.2604} C_DIS
LIN {X -42.4196,Y 88.7429,Z 101,A 110.0285,B 24.9187,C -2.0827,E1 24.9326,E2 335.3307} C_DIS
LIN {X -38.881,Y 90.3502,Z 101,A 107.967,B 24.9178,C -2.093,E1 24.9378,E2 337.3727} C_DIS
LIN {X -35.4582,Y 91.748,Z 101,A 105.5751,B 24.9183,C -2.0878,E1 24.9441,E2 339.7823} C_DIS
LIN {X -31.8845,Y 93.0494,Z 101,A 103.6837,B 24.9172,C -2.1017,E1 24.949,E2 341.6443} C_DIS
LIN {X -29.1167,Y 93.9515,Z 101,A 101.7129,B 24.9178,C -2.0942,E1 24.9543,E2 343.6365} C_DIS
LIN {X -26.2455,Y 94.7956,Z 101,A 100.121,B 24.9172,C -2.1013,E1 24.9585,E2 345.2141} C_DIS
LIN {X -23.1611,Y 95.5943,Z 101,A 98.1378,B 24.9174,C -2.0987,E1 24.9639,E2 347.2062} C_DIS
LIN {X -19.6567,Y 96.3759,Z 101,A 96.1073,B 24.9171,C -2.1026,E1 24.9694,E2 349.2299} C_DIS
LIN {X -16.2337,Y 97.011,Z 101,A 94.048,B 24.9171,C -2.1031,E1 24.9751,E2 351.2902} C_DIS
LIN {X -13.5929,Y 97.4165,Z 101,A 92.4785,B 24.9171,C -2.1036,E1 24.9794,E2 352.8597} C_DIS
LIN {X -8.8207,Y 97.9639,Z 101,A 89.75,B 24.9167,C -2.1076,E1 24.987,E2 355.5804} C_DIS
LIN {X -5.254,Y 98.2197,Z 101,A 87.7003,B 24.9165,C -2.1096,E1 24.9927,E2 357.6261} C_DIS
LIN {X -0.2769,Y 98.3601,Z 101,A 84.7903,B 24.9165,C -2.11,E1 25.0008,E2 360.5354} C_DIS
LIN {X 5.4539,Y 98.2086,Z 101,A 81.5561,B 24.9162,C -2.114,E1 25.0098,E2 363.7593} C_DIS
LIN {X 9.4432,Y 97.9064,Z 101,A 79.1292,B 24.9165,C -2.1104,E1 25.0166,E2 366.1934} C_DIS
LIN {X 12.2332,Y 97.5971,Z 101,A 77.2118,B 24.9173,C -2.1,E1 25.022,E2 368.1341} C_DIS
LIN {X 16.3477,Y 96.992,Z 101,A 74.963,B 24.9169,C -2.1055,E1 25.0281,E2 370.3677} C_DIS
LIN {X 19.8258,Y 96.3411,Z 101,A 72.8426,B 24.9171,C -2.1025,E1 25.0339,E2 372.4928} C_DIS
LIN {X 22.7396,Y 95.6971,Z 101,A 71.0458,B 24.9173,C -2.0994,E1 25.0388,E2 374.2944} C_DIS
LIN {X 26.5574,Y 94.7072,Z 101,A 68.825,B 24.9173,C -2.1007,E1 25.0448,E2 376.5086} C_DIS
LIN {X 33.4567,Y 92.4954,Z 101,A 64.7012,B 24.9173,C -2.1007,E1 25.0557,E2 380.6243} C_DIS
LIN {X 35.7012,Y 91.6525,Z 101,A 63.2226,B 24.9176,C -2.0964,E1 25.0596,E2 382.11} C_DIS
LIN {X 39.0546,Y 90.2745,Z 101,A 61.4548,B 24.9168,C -2.1069,E1 25.0641,E2 383.8489} C_DIS
LIN {X 41.5351,Y 89.16,Z 101,A 59.5869,B 24.9177,C -2.0945,E1 25.0689,E2 385.7414} C_DIS
LIN {X 44.8183,Y 87.5557,Z 101,A 57.4336,B 24.918,C -2.0909,E1 25.0743,E2 387.8974} C_DIS
LIN {X 47.9467,Y 85.8824,Z 101,A 55.3657,B 24.9182,C -2.0881,E1 25.0793,E2 389.9661} C_DIS
LIN {X 50.7246,Y 84.2726,Z 101,A 53.1778,B 24.9194,C -2.0735,E1 25.0847,E2 392.1818} C_DIS
LIN {X 54.3441,Y 81.9844,Z 101,A 50.9738,B 24.9188,C -2.0804,E1 25.0898,E2 394.3623} C_DIS
LIN {X 56.7779,Y 80.319,Z 101,A 49.5457,B 24.9182,C -2.0884,E1 25.093,E2 395.7666} C_DIS
LIN {X 59.136,Y 78.5978,Z 101,A 47.709,B 24.9188,C -2.0803,E1 25.0971,E2 397.6158} C_DIS
LIN {X 61.5218,Y 76.7465,Z 101,A 45.6641,B 24.9199,C -2.0662,E1 25.1017,E2 399.6863} C_DIS
LIN {X 64.7053,Y 74.0804,Z 101,A 43.4348,B 24.9197,C -2.0687,E1 25.1064,E2 401.901} C_DIS
LIN {X 67.3328,Y 71.7006,Z 101,A 41.3768,B 24.9201,C -2.0648,E1 25.1106,E2 403.96} C_DIS
LIN {X 69.9131,Y 69.187,Z 101,A 39.2927,B 24.9204,C -2.0609,E1 25.1147,E2 406.0445} C_DIS
LIN {X 72.3765,Y 66.6058,Z 101,A 37.2337,B 24.9207,C -2.057,E1 25.1187,E2 408.1037} C_DIS
LIN {X 74.8816,Y 63.7764,Z 101,A 35.0889,B 24.9209,C -2.0541,E1 25.1226,E2 410.2457} C_DIS
LIN {X 77.2532,Y 60.8822,Z 101,A 32.981,B 24.9211,C -2.0517,E1 25.1263,E2 412.3495} C_DIS
LIN {X 79.0347,Y 58.5534,Z 101,A 31.354,B 24.9211,C -2.0506,E1 25.129,E2 413.9713} C_DIS
LIN {X 81.8346,Y 54.5715,Z 101,A 28.2046,B 24.9226,C -2.0313,E1 25.1341,E2 417.1508} C_DIS
LIN {X 84.0928,Y 51.0205,Z 101,A 25.988,B 24.9224,C -2.034,E1 25.1373,E2 419.3498} C_DIS
LIN {X 85.6668,Y 48.3329,Z 101,A 24.0762,B 24.9231,C -2.0253,E1 25.14,E2 421.2723} C_DIS
LIN {X 87.409,Y 45.1053,Z 101,A 22.0465,B 24.9232,C -2.0236,E1 25.1426,E2 423.2953} C_DIS
LIN {X 88.6206,Y 42.6741,Z 101,A 20.6898,B 24.9229,C -2.0279,E1 25.1443,E2 424.6345} C_DIS
LIN {X 89.5727,Y 40.6383,Z 101,A 18.7339,B 24.9251,C -1.9991,E1 25.1466,E2 426.6479} C_DIS
LIN {X 90.8625,Y 37.6676,Z 101,A 17.0744,B 24.9248,C -2.0024,E1 25.1484,E2 428.2904} C_DIS
LIN {X 92.498,Y 33.4495,Z 101,A 14.5717,B 24.925,C -1.9998,E1 25.1508,E2 430.7853} C_DIS
LIN {X 93.6672,Y 30.0201,Z 101,A 12.657,B 24.925,C -2.0011,E1 25.1525,E2 432.6859} C_DIS
LIN {X 94.4315,Y 27.5242,Z 101,A 11.0499,B 24.9255,C -1.9931,E1 25.1538,E2 434.3027} C_DIS
LIN {X 95.2623,Y 24.4901,Z 101,A 9.2548,B 24.9258,C -1.989,E1 25.1551,E2 436.0973} C_DIS
LIN {X 96.0677,Y 21.1115,Z 101,A 7.2134,B 24.9263,C -1.982,E1 25.1563,E2 438.1433} C_DIS
LIN {X 96.7528,Y 17.7106,Z 101,A 5.0714,B 24.9272,C -1.971,E1 25.1575,E2 440.2989} C_DIS
LIN {X 97.3938,Y 13.7524,Z 101,A 2.3684,B 24.9288,C -1.9492,E1 25.1586,E2 443.0372} C_DIS
LIN {X 97.8332,Y 10.1663,Z 101,A 0.6866,B 24.928,C -1.9591,E1 25.1591,E2 444.6859} C_DIS
LIN {X 98.227,Y 5.1083,Z 101,A -2.2715,B 24.9287,C -1.9495,E1 25.1596,E2 447.649} C_DIS
LIN {X 98.3554,Y -1.0517,Z 101,A -5.6171,B 24.9289,C -1.9475,E1 25.1598,E2 450.9793} C_DIS
LIN {X 98.1964,Y -5.6755,Z 101,A -8.4656,B 24.93,C -1.9328,E1 25.1594,E2 453.8457} C_DIS
LIN {X 97.9373,Y -9.1081,Z 101,A -10.3059,B 24.93,C -1.9328,E1 25.159,E2 455.675} C_DIS
LIN {X 97.5935,Y -12.2607,Z 101,A -12.1936,B 24.9305,C -1.9252,E1 25.1584,E2 457.5694} C_DIS
LIN {X 97.1584,Y -15.3299,Z 101,A -14.119,B 24.9313,C -1.9147,E1 25.1576,E2 459.5083} C_DIS
LIN {X 96.5062,Y -19.0109,Z 101,A -15.9907,B 24.9309,C -1.9198,E1 25.1566,E2 461.3571} C_DIS
LIN {X 96.0057,Y -21.396,Z 101,A -17.6454,B 24.9319,C -1.906,E1 25.1556,E2 463.0348} C_DIS
LIN {X 95.1463,Y -24.9415,Z 101,A -19.7541,B 24.9323,C -1.8998,E1 25.1542,E2 465.1458} C_DIS
LIN {X 94.1617,Y -28.4336,Z 101,A -21.8322,B 24.9327,C -1.8946,E1 25.1526,E2 467.2245} C_DIS
LIN {X 92.9378,Y -32.2085,Z 101,A -23.9059,B 24.9326,C -1.8967,E1 25.1508,E2 469.2813} C_DIS
LIN {X 91.7637,Y -35.4181,Z 101,A -26.2059,B 24.9339,C -1.8784,E1 25.1485,E2 471.6118} C_DIS
LIN {X 90.3071,Y -38.9799,Z 101,A -28.3135,B 24.9339,C -1.8768,E1 25.1462,E2 473.7115} C_DIS
LIN {X 88.8627,Y -42.1702,Z 101,A -30.3592,B 24.9344,C -1.8704,E1 25.1438,E2 475.7612} C_DIS
LIN {X 87.3158,Y -45.2877,Z 101,A -32.4857,B 24.9351,C -1.8605,E1 25.1411,E2 477.8999} C_DIS
LIN {X 85.1349,Y -49.2626,Z 101,A -35.0955,B 24.9356,C -1.854,E1 25.1375,E2 480.5113} C_DIS
LIN {X 83.5034,Y -51.9797,Z 101,A -36.7153,B 24.9353,C -1.8576,E1 25.1352,E2 482.1144} C_DIS
LIN {X 81.7863,Y -54.6446,Z 101,A -38.6588,B 24.9359,C -1.8486,E1 25.1322,E2 484.0696} C_DIS
LIN {X 80.37,Y -56.7063,Z 101,A -40.1006,B 24.9362,C -1.8451,E1 25.1299,E2 485.5125} C_DIS
LIN {X 78.9377,Y -58.6836,Z 101,A -41.5952,B 24.9366,C -1.8384,E1 25.1274,E2 487.0158} C_DIS
LIN {X 76.8187,Y -61.4319,Z 101,A -43.9545,B 24.9379,C -1.8199,E1 25.1232,E2 489.4076} C_DIS
LIN {X 74.6824,Y -64.0102,Z 101,A -45.4553,B 24.9371,C -1.8323,E1 25.1206,E2 490.8724} C_DIS
LIN {X 72.6276,Y -66.3322,Z 101,A -47.2698,B 24.9374,C -1.8273,E1 25.1172,E2 492.6905} C_DIS
LIN {X 69.9043,Y -69.1959,Z 101,A -49.3291,B 24.9372,C -1.8311,E1 25.1132,E2 494.7321} C_DIS
LIN {X 66.7783,Y -72.2183,Z 101,A -52.0592,B 24.9381,C -1.8173,E1 25.1077,E2 497.4833} C_DIS
LIN {X 64.6074,Y -74.1659,Z 101,A -53.8386,B 24.9386,C -1.8103,E1 25.1039,E2 499.2722} C_DIS
LIN {X 61.822,Y -76.5032,Z 101,A -55.7554,B 24.9384,C -1.8134,E1 25.0998,E2 501.1746} C_DIS
LIN {X 58.9229,Y -78.7579,Z 101,A -58.0437,B 24.9391,C -1.8031,E1 25.0947,E2 503.4789} C_DIS
LIN {X 55.9923,Y -80.8676,Z 101,A -59.9927,B 24.939,C -1.8047,E1 25.0903,E2 505.4173} C_DIS
LIN {X 53.5237,Y -82.5234,Z 101,A -61.9874,B 24.9399,C -1.7912,E1 25.0856,E2 507.4373} C_DIS
LIN {X 50.7778,Y -84.2403,Z 101,A -64.0471,B 24.9405,C -1.7811,E1 25.0806,E2 509.5144} C_DIS
LIN {X 47.1561,Y -86.3195,Z 101,A -66.0708,B 24.9398,C -1.7923,E1 25.0757,E2 511.5057} C_DIS
LIN {X 44.3152,Y -87.8128,Z 101,A -68.0543,B 24.9403,C -1.7848,E1 25.0708,E2 513.5014} C_DIS
LIN {X 41.3171,Y -89.2615,Z 101,A -69.8394,B 24.9401,C -1.7876,E1 25.0663,E2 515.2753} C_DIS
LIN {X 38.3033,Y -90.5955,Z 101,A -72.0197,B 24.941,C -1.7749,E1 25.0607,E2 517.4803} C_DIS
LIN {X 34.2546,Y -92.2043,Z 101,A -74.3783,B 24.9407,C -1.7782,E1 25.0545,E2 519.8261} C_DIS
LIN {X 31.8621,Y -93.0575,Z 101,A -75.9656,B 24.9411,C -1.7722,E1 25.0503,E2 521.4243} C_DIS
LIN {X 28.0919,Y -94.2631,Z 101,A -78.0858,B 24.9408,C -1.7765,E1 25.0447,E2 523.5306} C_DIS
LIN {X 24.7489,Y -95.1958,Z 101,A -80.1228,B 24.941,C -1.7738,E1 25.0392,E2 525.5708} C_DIS
LIN {X 20.9994,Y -96.0922,Z 101,A -82.307,B 24.941,C -1.7739,E1 25.0333,E2 527.7516} C_DIS
LIN {X 18.0177,Y -96.6974,Z 101,A -84.4307,B 24.942,C -1.7594,E1 25.0274,E2 529.9073} C_DIS
LIN {X 13.3356,Y -97.453,Z 101,A -86.9533,B 24.9415,C -1.7663,E1 25.0204,E2 532.4112} C_DIS
LIN {X 7.8656,Y -98.0449,Z 101,A -90.016,B 24.9413,C -1.7698,E1 25.012,E2 535.4636} C_DIS
LIN {X 3.6596,Y -98.2929,Z 101,A -92.7963,B 24.9421,C -1.7569,E1 25.0041,E2 538.2736} C_DIS
LIN {X 0.7034,Y -98.3509,Z 101,A -94.9031,B 24.9431,C -1.7427,E1 24.9982,E2 540.4139} C_DIS
Enddeposition()
LIN {X 0.7034,Y -98.3509,Z 101,A -94.9031,B 24.9431,C -1.7427,E1 24.9982,E2 540.4139} C_DIS
Startdeposition()
$VEL.CP = VEL_PRINT
LIN {X 2.0004,Y -97.4698,Z 101,A -92.7062,B 24.9386,C -1.8102,E1 25.0047,E2 538.0571} C_DIS
LIN {X 4.6843,Y -97.3788,Z 101,A -91.1771,B 24.9386,C -1.809,E1 25.009,E2 536.5314} C_DIS
LIN {X 7.0171,Y -97.2383,Z 101,A -89.8058,B 24.9386,C -1.8095,E1 25.0128,E2 535.1594} C_DIS
LIN {X 9.3291,Y -97.0434,Z 101,A -88.4672,B 24.9386,C -1.8093,E1 25.0165,E2 533.8221} C_DIS
LIN {X 11.9328,Y -96.7589,Z 101,A -86.9064,B 24.9386,C -1.811,E1 25.0209,E2 532.2584} C_DIS
LIN {X 14.2935,Y -96.4384,Z 101,A -85.5085,B 24.9385,C -1.8119,E1 25.0247,E2 530.8597} C_DIS
LIN {X 16.6449,Y -96.0604,Z 101,A -84.111,B 24.9384,C -1.8129,E1 25.0286,E2 529.4613} C_DIS
LIN {X 18.8538,Y -95.6506,Z 101,A -82.7853,B 24.9384,C -1.8142,E1 25.0322,E2 528.134} C_DIS
LIN {X 21.3019,Y -95.1359,Z 101,A -81.3248,B 24.9382,C -1.8152,E1 25.0362,E2 526.6731} C_DIS
LIN {X 23.689,Y -94.5702,Z 101,A -79.8873,B 24.9382,C -1.8164,E1 25.0401,E2 525.2347} C_DIS
LIN {X 27.1436,Y -93.637,Z 101,A -77.7891,B 24.938,C -1.8185,E1 25.0458,E2 523.135} C_DIS
LIN {X 29.4262,Y -92.9449,Z 101,A -76.391,B 24.938,C -1.82,E1 25.0495,E2 521.7358} C_DIS
LIN {X 31.6901,Y -92.1976,Z 101,A -74.995,B 24.9378,C -1.8216,E1 25.0532,E2 520.3389} C_DIS
LIN {X 33.9217,Y -91.3999,Z 101,A -73.6045,B 24.9377,C -1.8233,E1 25.0568,E2 518.947} C_DIS
LIN {X 36.1519,Y -90.541,Z 101,A -72.2071,B 24.9376,C -1.825,E1 25.0605,E2 517.5488} C_DIS
LIN {X 38.422,Y -89.6015,Z 101,A -70.7713,B 24.9374,C -1.8268,E1 25.0642,E2 516.1121} C_DIS
LIN {X 40.6023,Y -88.6348,Z 101,A -69.3701,B 24.9373,C -1.829,E1 25.0677,E2 514.7093} C_DIS
LIN {X 43.7854,Y -87.106,Z 101,A -67.3,B 24.9371,C -1.8321,E1 25.0729,E2 512.6372} C_DIS
LIN {X 45.9028,Y -86.009,Z 101,A -65.9035,B 24.9369,C -1.8343,E1 25.0764,E2 511.2394} C_DIS
LIN {X 48.0324,Y -84.8383,Z 101,A -64.4809,B 24.9368,C -1.8366,E1 25.0799,E2 509.8156} C_DIS
LIN {X 50.0909,Y -83.6394,Z 101,A -63.0891,B 24.9366,C -1.8389,E1 25.0832,E2 508.4227} C_DIS
LIN {X 52.1338,Y -82.3815,Z 101,A -61.6822,B 24.9364,C -1.8415,E1 25.0866,E2 507.0142} C_DIS
LIN {X 54.1708,Y -81.0568,Z 101,A -60.2625,B 24.9363,C -1.844,E1 25.0899,E2 505.5933} C_DIS
LIN {X 56.0989,Y -79.7342,Z 101,A -58.8913,B 24.9361,C -1.8466,E1 25.093,E2 504.2205} C_DIS
LIN {X 58.0694,Y -78.311,Z 101,A -57.2578,B 24.9353,C -1.8576,E1 25.0967,E2 502.567} C_DIS
LIN {X 60.9003,Y -76.1302,Z 101,A -55.1641,B 24.935,C -1.8619,E1 25.1013,E2 500.4709} C_DIS
LIN {X 63.6692,Y -73.8302,Z 101,A -53.0649,B 24.9347,C -1.866,E1 25.1058,E2 498.37} C_DIS
LIN {X 66.3441,Y -71.4362,Z 101,A -50.9648,B 24.9344,C -1.8706,E1 25.1101,E2 496.2676} C_DIS
LIN {X 68.9372,Y -68.9372,Z 101,A -48.8561,B 24.9341,C -1.8754,E1 25.1143,E2 494.1564} C_DIS
LIN {X 71.4356,Y -66.3448,Z 101,A -46.7554,B 24.9337,C -1.8801,E1 25.1184,E2 492.0537} C_DIS
LIN {X 73.8001,Y -63.7039,Z 101,A -44.681,B 24.9334,C -1.8851,E1 25.1222,E2 489.9769} C_DIS
LIN {X 76.1086,Y -60.9274,Z 101,A -42.569,B 24.933,C -1.8903,E1 25.1259,E2 487.8623} C_DIS
LIN {X 78.3105,Y -58.0701,Z 101,A -40.6798,B 24.9332,C -1.887,E1 25.1291,E2 485.99} C_DIS
LIN {X 79.6807,Y -56.1748,Z 101,A -39.3087,B 24.933,C -1.8907,E1 25.1313,E2 484.6169} C_DIS
LIN {X 81.031,Y -54.2088,Z 101,A -37.9165,B 24.9327,C -1.8942,E1 25.1335,E2 483.2232} C_DIS
LIN {X 82.3575,Y -52.1718,Z 101,A -36.4979,B 24.9325,C -1.8979,E1 25.1356,E2 481.8031} C_DIS
LIN {X 83.5519,Y -50.2356,Z 101,A -35.1747,B 24.9322,C -1.9012,E1 25.1376,E2 480.4789} C_DIS
LIN {X 84.5951,Y -48.4564,Z 101,A -33.8923,B 24.9318,C -1.9075,E1 25.1394,E2 479.1882} C_DIS
LIN {X 85.9862,Y -45.9461,Z 101,A -32.2891,B 24.9317,C -1.9091,E1 25.1415,E2 477.5896} C_DIS
LIN {X 87.0848,Y -43.8283,Z 101,A -30.8961,B 24.9314,C -1.9129,E1 25.1433,E2 476.195} C_DIS
LIN {X 88.1112,Y -41.7258,Z 101,A -29.5281,B 24.9311,C -1.9168,E1 25.1449,E2 474.8252} C_DIS
LIN {X 89.1059,Y -39.5571,Z 101,A -28.1341,B 24.9308,C -1.9207,E1 25.1465,E2 473.4295} C_DIS
LIN {X 90.047,Y -37.365,Z 101,A -26.7414,B 24.9306,C -1.9246,E1 25.148,E2 472.0352} C_DIS
LIN {X 90.9509,Y -35.1082,Z 101,A -25.3266,B 24.9303,C -1.9285,E1 25.1495,E2 470.6191} C_DIS
LIN {X 91.7925,Y -32.8453,Z 101,A -23.9137,B 24.93,C -1.9326,E1 25.1508,E2 469.2044} C_DIS
LIN {X 92.5331,Y -30.6949,Z 101,A -22.573,B 24.9297,C -1.937,E1 25.152,E2 467.8609} C_DIS
LIN {X 93.2835,Y -28.3343,Z 101,A -21.1357,B 24.9294,C -1.9408,E1 25.1532,E2 466.4228} C_DIS
LIN {X 93.9056,Y -26.1959,Z 101,A -19.8242,B 24.9291,C -1.9451,E1 25.1542,E2 465.1087} C_DIS
LIN {X 94.5698,Y -23.6902,Z 101,A -18.328,B 24.9288,C -1.9488,E1 25.1553,E2 463.6123} C_DIS
LIN {X 95.3757,Y -20.2024,Z 101,A -16.2369,B 24.9283,C -1.955,E1 25.1565,E2 461.5187} C_DIS
LIN {X 95.8358,Y -17.8922,Z 101,A -14.8635,B 24.928,C -1.9591,E1 25.1573,E2 460.1438} C_DIS
LIN {X 96.2004,Y -15.8078,Z 101,A -13.5877,B 24.9277,C -1.9643,E1 25.1579,E2 458.8631} C_DIS
LIN {X 96.5989,Y -13.1638,Z 101,A -12.069,B 24.9274,C -1.9673,E1 25.1585,E2 457.3464} C_DIS
LIN {X 96.8919,Y -10.7977,Z 101,A -10.6754,B 24.9271,C -1.9715,E1 25.1589,E2 455.9511} C_DIS
LIN {X 97.1269,Y -8.4254,Z 101,A -9.2854,B 24.9268,C -1.9756,E1 25.1593,E2 454.5596} C_DIS
LIN {X 97.3068,Y -6.0029,Z 101,A -7.8681,B 24.9265,C -1.9798,E1 25.1595,E2 453.1408} C_DIS
LIN {X 97.4243,Y -3.6248,Z 101,A -6.478,B 24.9262,C -1.984,E1 25.1597,E2 451.7492} C_DIS
LIN {X 97.4844,Y -1.2066,Z 101,A -5.0679,B 24.9259,C -1.9881,E1 25.1597,E2 450.3377} C_DIS
LIN {X 97.4853,Y 1.0893,Z 101,A -3.725,B 24.9256,C -1.9922,E1 25.1597,E2 448.9931} C_DIS
LIN {X 97.4279,Y 3.5243,Z 101,A -2.307,B 24.9253,C -1.9963,E1 25.1597,E2 447.5739} C_DIS
LIN {X 97.3146,Y 5.8675,Z 101,A -0.9404,B 24.925,C -2.0002,E1 25.1594,E2 446.2062} C_DIS
LIN {X 97.1582,Y 8.0432,Z 101,A 0.3717,B 24.9246,C -2.0055,E1 25.1591,E2 444.8893} C_DIS
LIN {X 96.9079,Y 10.6509,Z 101,A 1.8671,B 24.9243,C -2.0087,E1 25.1587,E2 443.3955} C_DIS
LIN {X 96.6196,Y 13.0082,Z 101,A 3.2364,B 24.9241,C -2.012,E1 25.1582,E2 442.0262} C_DIS
LIN {X 96.2622,Y 15.4343,Z 101,A 4.6848,B 24.9237,C -2.0169,E1 25.1576,E2 440.5749} C_DIS
LIN {X 95.8748,Y 17.6787,Z 101,A 6.0259,B 24.9234,C -2.0212,E1 25.1569,E2 439.2316} C_DIS
LIN {X 95.3876,Y 20.1453,Z 101,A 7.4809,B 24.9231,C -2.0249,E1 25.1561,E2 437.7763} C_DIS
LIN {X 94.8556,Y 22.5187,Z 101,A 8.901,B 24.9228,C -2.0289,E1 25.1552,E2 436.3549} C_DIS
LIN {X 94.2877,Y 24.7881,Z 101,A 10.2665,B 24.9225,C -2.0328,E1 25.1543,E2 434.9881} C_DIS
LIN {X 93.7263,Y 26.8284,Z 101,A 11.5378,B 24.9221,C -2.0377,E1 25.1533,E2 433.7126} C_DIS
LIN {X 92.9397,Y 29.4432,Z 101,A 13.0962,B 24.9219,C -2.0407,E1 25.152,E2 432.156} C_DIS
LIN {X 92.1905,Y 31.7111,Z 101,A 14.4909,B 24.9216,C -2.0445,E1 25.1508,E2 430.7601} C_DIS
LIN {X 91.4019,Y 33.9162,Z 101,A 15.8579,B 24.9213,C -2.0482,E1 25.1495,E2 429.392} C_DIS
LIN {X 90.5533,Y 36.1205,Z 101,A 17.2353,B 24.9211,C -2.0519,E1 25.1481,E2 428.0137} C_DIS
LIN {X 89.6787,Y 38.239,Z 101,A 18.5568,B 24.9208,C -2.0548,E1 25.1467,E2 426.6925} C_DIS
LIN {X 88.6381,Y 40.5951,Z 101,A 20.0847,B 24.9205,C -2.0596,E1 25.1449,E2 425.1615} C_DIS
LIN {X 87.6117,Y 42.7653,Z 101,A 21.4809,B 24.9202,C -2.063,E1 25.1432,E2 423.7648} C_DIS
LIN {X 86.5597,Y 44.8558,Z 101,A 22.8502,B 24.9199,C -2.0666,E1 25.1415,E2 422.3943} C_DIS
LIN {X 85.4357,Y 46.9612,Z 101,A 24.2454,B 24.9196,C -2.0701,E1 25.1396,E2 420.9981} C_DIS
LIN {X 84.2143,Y 49.1181,Z 101,A 25.8978,B 24.9187,C -2.0817,E1 25.1373,E2 419.327} C_DIS
LIN {X 82.391,Y 52.1186,Z 101,A 27.7438,B 24.919,C -2.0786,E1 25.1346,E2 417.4975} C_DIS
LIN {X 81.0621,Y 54.1628,Z 101,A 29.1694,B 24.9187,C -2.082,E1 25.1324,E2 416.071} C_DIS
LIN {X 79.7483,Y 56.0787,Z 101,A 30.5283,B 24.9185,C -2.0853,E1 25.1302,E2 414.7111} C_DIS
LIN {X 78.3066,Y 58.0755,Z 101,A 32.1752,B 24.9176,C -2.0966,E1 25.1275,E2 413.0454} C_DIS
LIN {X 76.1346,Y 60.8947,Z 101,A 34.2622,B 24.9172,C -2.1014,E1 25.1239,E2 410.9568} C_DIS
LIN {X 73.8365,Y 63.6618,Z 101,A 36.3634,B 24.9168,C -2.1058,E1 25.1201,E2 408.8548} C_DIS
LIN {X 71.4238,Y 66.3575,Z 101,A 38.4797,B 24.9165,C -2.1102,E1 25.1161,E2 406.7374} C_DIS
LIN {X 68.937,Y 68.9373,Z 101,A 40.5694,B 24.9162,C -2.1141,E1 25.112,E2 404.6473} C_DIS
LIN {X 66.3572,Y 71.4241,Z 101,A 42.6728,B 24.9158,C -2.1184,E1 25.1077,E2 402.5426} C_DIS
LIN {X 63.6872,Y 73.8147,Z 101,A 44.7719,B 24.9155,C -2.1222,E1 25.1033,E2 400.4426} C_DIS
LIN {X 60.9106,Y 76.122,Z 101,A 46.8759,B 24.9153,C -2.1256,E1 25.0987,E2 398.3388} C_DIS
LIN {X 58.0733,Y 78.3082,Z 101,A 48.7647,B 24.9156,C -2.1211,E1 25.0946,E2 396.4673} C_DIS
LIN {X 56.1756,Y 79.6802,Z 101,A 50.1386,B 24.9154,C -2.1234,E1 25.0914,E2 395.0928} C_DIS
LIN {X 54.2071,Y 81.0322,Z 101,A 51.536,B 24.9153,C -2.1255,E1 25.0882,E2 393.6952} C_DIS
LIN {X 52.164,Y 82.3625,Z 101,A 52.964,B 24.9151,C -2.1275,E1 25.0849,E2 392.267} C_DIS
LIN {X 50.1862,Y 83.5819,Z 101,A 54.3162,B 24.915,C -2.1291,E1 25.0816,E2 390.9154} C_DIS
LIN {X 48.0985,Y 84.8007,Z 101,A 55.7415,B 24.9148,C -2.1313,E1 25.0782,E2 389.4892} C_DIS
LIN {X 45.9865,Y 85.9645,Z 101,A 57.1578,B 24.9147,C -2.1332,E1 25.0747,E2 388.0724} C_DIS
LIN {X 43.8311,Y 87.0834,Z 101,A 58.5762,B 24.9145,C -2.1347,E1 25.0712,E2 386.6544} C_DIS
LIN {X 41.7279,Y 88.1102,Z 101,A 59.9497,B 24.9145,C -2.1363,E1 25.0677,E2 385.2807} C_DIS
LIN {X 39.5585,Y 89.1052,Z 101,A 61.3498,B 24.9143,C -2.1378,E1 25.0642,E2 383.8805} C_DIS
LIN {X 37.3658,Y 90.0467,Z 101,A 62.749,B 24.9142,C -2.1392,E1 25.0606,E2 382.4813} C_DIS
LIN {X 35.1083,Y 90.9509,Z 101,A 64.1735,B 24.9141,C -2.1404,E1 25.0569,E2 381.057} C_DIS
LIN {X 33.0816,Y 91.7063,Z 101,A 65.4579,B 24.9139,C -2.1421,E1 25.0535,E2 379.7713} C_DIS
LIN {X 30.7161,Y 92.526,Z 101,A 66.9108,B 24.9139,C -2.1427,E1 25.0496,E2 378.3199} C_DIS
LIN {X 28.5694,Y 93.2106,Z 101,A 68.2622,B 24.9137,C -2.1447,E1 25.046,E2 376.9661} C_DIS
LIN {X 26.0504,Y 93.9468,Z 101,A 69.7713,B 24.9137,C -2.1445,E1 25.042,E2 375.46} C_DIS
LIN {X 23.6962,Y 94.5683,Z 101,A 71.2023,B 24.9137,C -2.1454,E1 25.0381,E2 374.0291} C_DIS
LIN {X 21.4179,Y 95.1099,Z 101,A 72.5782,B 24.9137,C -2.1461,E1 25.0344,E2 372.6534} C_DIS
LIN {X 19.0174,Y 95.6191,Z 101,A 74.0168,B 24.9136,C -2.1466,E1 25.0304,E2 371.2154} C_DIS
LIN {X 16.7168,Y 96.0478,Z 101,A 75.3911,B 24.9136,C -2.1471,E1 25.0267,E2 369.8414} C_DIS
LIN {X 14.3151,Y 96.4352,Z 101,A 76.8209,B 24.9135,C -2.1476,E1 25.0227,E2 368.4119} C_DIS
LIN {X 12.0293,Y 96.7464,Z 101,A 78.178,B 24.9135,C -2.1479,E1 25.019,E2 367.0551} C_DIS
LIN {X 9.5677,Y 97.0213,Z 101,A 79.6311,B 24.9135,C -2.148,E1 25.0149,E2 365.6027} C_DIS
LIN {X 7.2413,Y 97.2223,Z 101,A 81.0047,B 24.9135,C -2.1481,E1 25.0111,E2 364.2295} C_DIS
LIN {X 3.6124,Y 97.4249,Z 101,A 83.1393,B 24.9135,C -2.1481,E1 25.0052,E2 362.0959} C_DIS
LIN {X 1.2462,Y 97.4837,Z 101,A 84.53,B 24.9135,C -2.1478,E1 25.0013,E2 360.7058} C_DIS
LIN {X -1.1099,Y 97.4852,Z 101,A 85.9138,B 24.9135,C -2.1475,E1 24.9974,E2 359.3229} C_DIS
LIN {X -3.4361,Y 97.4306,Z 101,A 87.2918,B 24.9135,C -2.1475,E1 24.9936,E2 357.9447} C_DIS
LIN {X -5.969,Y 97.309,Z 101,A 88.7763,B 24.9135,C -2.1467,E1 24.9894,E2 356.4616} C_DIS
LIN {X -8.3415,Y 97.1343,Z 101,A 90.1761,B 24.9136,C -2.1461,E1 24.9855,E2 355.0625} C_DIS
LIN {X -10.6606,Y 96.9069,Z 101,A 91.5486,B 24.9136,C -2.1455,E1 24.9817,E2 353.6907} C_DIS
LIN {X -13.0601,Y 96.6129,Z 101,A 92.9584,B 24.9138,C -2.1443,E1 24.9778,E2 352.2828} C_DIS
LIN {X -15.4386,Y 96.2615,Z 101,A 94.386,B 24.9138,C -2.1438,E1 24.9739,E2 350.855} C_DIS
LIN {X -17.8356,Y 95.8466,Z 101,A 95.8171,B 24.9138,C -2.1428,E1 24.97,E2 349.425} C_DIS
LIN {X -20.1302,Y 95.3907,Z 101,A 97.1947,B 24.914,C -2.1417,E1 24.9662,E2 348.0483} C_DIS
LIN {X -22.2369,Y 94.9207,Z 101,A 98.4971,B 24.914,C -2.1417,E1 24.9626,E2 346.7441} C_DIS
LIN {X -24.4773,Y 94.3675,Z 101,A 99.8703,B 24.914,C -2.141,E1 24.9589,E2 345.3706} C_DIS
LIN {X -27.1517,Y 93.6347,Z 101,A 101.4583,B 24.9143,C -2.1378,E1 24.9547,E2 343.7877} C_DIS
LIN {X -30.5289,Y 92.5884,Z 101,A 103.5425,B 24.9145,C -2.1357,E1 24.9491,E2 341.705} C_DIS
LIN {X -32.8309,Y 91.7976,Z 101,A 104.9758,B 24.9145,C -2.134,E1 24.9454,E2 340.2729} C_DIS
LIN {X -35.0252,Y 90.9826,Z 101,A 106.3329,B 24.9148,C -2.1315,E1 24.9418,E2 338.9189} C_DIS
LIN {X -38.4214,Y 89.6017,Z 101,A 108.5111,B 24.915,C -2.1293,E1 24.9362,E2 336.7411} C_DIS
LIN {X -40.6044,Y 88.6338,Z 101,A 109.9239,B 24.9151,C -2.1275,E1 24.9326,E2 335.3291} C_DIS
LIN {X -42.7633,Y 87.6126,Z 101,A 111.3327,B 24.9153,C -2.1255,E1 24.9291,E2 333.9214} C_DIS
LIN {X -44.8443,Y 86.5656,Z 101,A 112.708,B 24.9154,C -2.1234,E1 24.9256,E2 332.5473} C_DIS
LIN {X -46.9621,Y 85.4352,Z 101,A 114.1249,B 24.9156,C -2.1213,E1 24.9222,E2 331.1316} C_DIS
LIN {X -49.0808,Y 84.2363,Z 101,A 115.56,B 24.9158,C -2.1189,E1 24.9187,E2 329.6979} C_DIS
LIN {X -51.1501,Y 82.996,Z 101,A 116.9791,B 24.916,C -2.1163,E1 24.9153,E2 328.2804} C_DIS
LIN {X -53.1244,Y 81.7461,Z 101,A 118.3636,B 24.9162,C -2.1141,E1 24.9121,E2 326.8968} C_DIS
LIN {X -55.1447,Y 80.3974,Z 101,A 119.7962,B 24.9164,C -2.1114,E1 24.9088,E2 325.4658} C_DIS
LIN {X -57.0924,Y 79.026,Z 101,A 121.2027,B 24.9166,C -2.1088,E1 24.9056,E2 324.0606} C_DIS
LIN {X -59.0046,Y 77.6087,Z 101,A 122.8179,B 24.9163,C -2.1132,E1 24.9019,E2 322.4292} C_DIS
LIN {X -61.8276,Y 75.3791,Z 101,A 124.9449,B 24.9166,C -2.109,E1 24.8973,E2 320.3041} C_DIS
LIN {X -64.5167,Y 73.0902,Z 101,A 127.0183,B 24.917,C -2.1043,E1 24.8929,E2 318.2339} C_DIS
LIN {X -67.0803,Y 70.744,Z 101,A 129.0016,B 24.9175,C -2.0975,E1 24.8889,E2 316.2586} C_DIS
LIN {X -69.5304,Y 68.3367,Z 101,A 130.9374,B 24.9181,C -2.0899,E1 24.8851,E2 314.3327} C_DIS
LIN {X -71.7357,Y 66.0176,Z 101,A 132.914,B 24.9182,C -2.0884,E1 24.8813,E2 312.351} C_DIS
LIN {X -74.2016,Y 63.2333,Z 101,A 135,B 24.9189,C -2.0795,E1 24.8775,E2 310.2768} C_DIS
LIN {X -76.1247,Y 60.9072,Z 101,A 136.9791,B 24.9187,C -2.0817,E1 24.874,E2 308.2834} C_DIS
LIN {X -78.2966,Y 58.0887,Z 101,A 138.8772,B 24.9197,C -2.0696,E1 24.8708,E2 306.4049} C_DIS
LIN {X -79.6587,Y 56.2057,Z 101,A 140.2528,B 24.9199,C -2.0662,E1 24.8686,E2 305.0307} C_DIS
LIN {X -80.9973,Y 54.2586,Z 101,A 141.6519,B 24.9202,C -2.0627,E1 24.8664,E2 303.633} C_DIS
LIN {X -82.6808,Y 51.6547,Z 101,A 143.5865,B 24.9203,C -2.0613,E1 24.8635,E2 301.6919} C_DIS
LIN {X -84.2041,Y 49.1355,Z 101,A 145.2235,B 24.9209,C -2.0533,E1 24.8612,E2 300.0657} C_DIS
LIN {X -85.3482,Y 47.1194,Z 101,A 146.6002,B 24.9212,C -2.0498,E1 24.8593,E2 298.6901} C_DIS
LIN {X -86.528,Y 44.9172,Z 101,A 148.0724,B 24.9215,C -2.0456,E1 24.8574,E2 297.2201} C_DIS
LIN {X -87.4574,Y 43.0766,Z 101,A 149.3312,B 24.9217,C -2.0436,E1 24.8558,E2 295.9594} C_DIS
LIN {X -88.6162,Y 40.6423,Z 101,A 150.8872,B 24.9221,C -2.0379,E1 24.854,E2 294.4085} C_DIS
LIN {X -89.6039,Y 38.4164,Z 101,A 152.3276,B 24.9224,C -2.0338,E1 24.8524,E2 292.9697} C_DIS
LIN {X -90.5277,Y 36.1855,Z 101,A 153.9203,B 24.9224,C -2.0352,E1 24.8507,E2 291.3649} C_DIS
LIN {X -91.6115,Y 33.3416,Z 101,A 155.6388,B 24.9229,C -2.0274,E1 24.8491,E2 289.6554} C_DIS
LIN {X -92.5498,Y 30.6453,Z 101,A 157.2479,B 24.9235,C -2.0199,E1 24.8476,E2 288.055} C_DIS
LIN {X -93.2689,Y 28.3814,Z 101,A 158.8629,B 24.9233,C -2.0227,E1 24.8463,E2 286.424} C_DIS
LIN {X -94.2427,Y 24.9572,Z 101,A 161.0012,B 24.9237,C -2.0176,E1 24.8447,E2 284.2853} C_DIS
LIN {X -94.9618,Y 22.0589,Z 101,A 162.5852,B 24.9245,C -2.0064,E1 24.8437,E2 282.7187} C_DIS
LIN {X -95.6207,Y 19.0092,Z 101,A 164.3672,B 24.9251,C -1.9989,E1 24.8427,E2 280.9443} C_DIS
LIN {X -96.0496,Y 16.7067,Z 101,A 165.7593,B 24.9254,C -1.995,E1 24.842,E2 279.5532} C_DIS
LIN {X -96.4371,Y 14.3028,Z 101,A 167.1995,B 24.9257,C -1.9907,E1 24.8414,E2 278.1147} C_DIS
Enddeposition()
END
